EQUIP_TYPE_5_xv501a(
	i1:=NOT sludge_holding_A.q3  OR hold_thickening_process ,
	i2:= sludge_holding_A.q3,
	sa1:=XV505A_SolenoidValveLine_CloseStat ,
	sa2:=XV505A_SolenoidValveLine_OpenStat ,
	c1=> ,
	q1=>XV505A_SolenoidValveLine_OpenCmd ,
	e1=> );
EQUIP_TYPE_5_xv501b(
	i1:=NOT sludge_holding_A.q4  OR hold_thickening_process ,
	i2:= sludge_holding_A.q4,
	sa1:=XV501A_AirBlowerValve_CloseStat ,
	sa2:=XV501A_AirBlowerValve_OpenStat ,
	c1=> ,
	q1=>XV501A_AirBlowerValve_OpenCmd ,
	e1=> );

EQUIP_TYPE_4_d503(
	i1:=NOT sludge_holding_A.q5  OR hold_thickening_process ,
	i2:= sludge_holding_A.q5,
	sa1:= D503A_DrumThickener_EStopStat,
	sa2:= D503A_DrumThickener_LocalRemoteStat,
	sa3:= D503A_DrumThickener_OverloadStat,
	sa4:= D503A_DrumThickener_RunStat,
	c1=> ,
	q1=> D503A_DrumThickener_RunCmd );

EQUP_TYPE_1_p505(
	i1:=NOT sludge_holding_A.q6  OR hold_thickening_process ,
	i2:=sludge_holding_A.q6 ,
	r1:=reset_p505 ,
	sa1:= P505A_BackwashWaterPump_EStopStat,
	sa2:= ,
	sa3:= P505A_BackwashWaterPump_LocalRemoteStat,
	sa4:= P505A_BackwashWaterPump_OverloadStat ,
	sa5:= P505A_BackwashWaterPump_RunStat,
	sb1:= P505B_BackwashWaterPump_EStopStat,
	sb2:= ,
	sb3:= P505B_BackwashWaterPump_LocalRemoteStat,
	sb4:= P505B_BackwashWaterPump_OverloadStat ,
	sb5:= P505B_BackwashWaterPump_RunStat,
	c1=> ,
	c2=> ,
	q1=>P505A_BackwashWaterPump_RunCmd ,
	q2=>P505B_BackwashWaterPump_RunCmd ,
	e1=> );

EQUIP_TYPE_5_xv505A(
	i1:=NOT sludge_holding_A.q7  OR hold_thickening_process ,
	i2:=sludge_holding_A.q7 ,
	sa1:= XV505A_SolenoidValveLine_CloseStat,
	sa2:= XV505A_SolenoidValveLine_OpenStat,
	c1=> ,
	q1=> XV505A_SolenoidValveLine_OpenCmd,
	e1=> );
EQUIP_TYPE_5_xv505B(
	i1:=NOT sludge_holding_A.q7  OR hold_thickening_process ,
	i2:=sludge_holding_A.q7 ,
	sa1:= XV505B_SolenoidValveLine_CloseStat,
	sa2:= XV505B_SolenoidValveLine_OpenStat,
	c1=> ,
	q1=> XV505B_SolenoidValveLine_CloseCmd,
	e1=> );
EQUIP_TYPE_4_M502A(
	i1:= NOT sludge_holding_A.q8  OR hold_thickening_process,
	i2:= sludge_holding_A.q8,
	sa1:= M502A_Floculator_EStopStat,
	sa2:= M502A_Floculator_LocalRemoteStat,
	sa3:= M502A_Floculator_OverloadStat,
	sa4:= M502A_Floculator_RunStat,
	c1=> ,
	q1=> M502A_Floculator_RunCmd,
	e1=> );
EQUIP_TYPE_4_M502B(
	i1:= NOT sludge_holding_A.q8  OR hold_thickening_process,
	i2:= sludge_holding_A.q8,
	sa1:= M502B_Floculator_EStopStat,
	sa2:= M502B_Floculator_LocalRemoteStat,
	sa3:= M502B_Floculator_OverloadStat,
	sa4:= M502B_Floculator_RunStat,
	c1=> ,
	q1=> M502B_Floculator_RunCmd,
	e1=> );

EQUIPMENT_REDUNDANT_AIRBLOWER_p501(
	i1:= sludge_holding_A.q9_1A  OR hold_thickening_process ,
	i2:= sludge_holding_A.q9_2A,
	i3:= sludge_holding_A.q9_1B  OR hold_thickening_process,
	i4:= sludge_holding_A.q9_2B,
	sa1:= P501A_SludgeFeedPump_EStopStat ,
	sa2:= P501A_SludgeFeedPump_IncompleteStat,
	sa3:= P501A_SludgeFeedPump_LocalRemoteStat,
	sa4:= P501A_SludgeFeedPump_OverloadStat,
	sa5:= P501A_SludgeFeedPump_RunStat,
	sb1:= P501B_SludgeFeedPump_EStopStat ,
	sb2:= P501B_SludgeFeedPump_IncompleteStat,
	sb3:= P501B_SludgeFeedPump_LocalRemoteStat,
	sb4:= P501B_SludgeFeedPump_OverloadStat,
	sb5:= P501B_SludgeFeedPump_RunStat,
	sc1:= P501C_SludgeFeedPump_EStopStat ,
	sc2:= P501C_SludgeFeedPump_IncompleteStat,
	sc3:= P501C_SludgeFeedPump_LocalRemoteStat,
	sc4:= P501C_SludgeFeedPumpOverloadStat,
	sc5:= P501C_SludgeFeedPump_RunStat,
	r1 := reset_p501,
	q1=> P501A_SludgeFeedPump_RunCmd,
	q2=> P501B_SludgeFeedPump_RunCmd,
	q3=> P501C_SludgeFeedPump_RunCmd,
	e1=>);

EQUIP_TYPE_5_XVPolymerWaterSupply(
	i1:= sludge_holding_A.q10  OR hold_thickening_process,
	i2:= sludge_holding_A.q11,
	sa1:= XVW501A_WaterValve_CloseStat,
	sa2:= XVW501A_WaterValve_OpenStat ,
	c1=> ,
	q1=> XVW501A_WaterValve_OpenCmd,
	e1=> );

EQUIP_STIRRER_M503(
	i1:= NOT sludge_holding_A.q12  OR hold_thickening_process,
	i2:= sludge_holding_A.q12,
	sa1:= M503_PolymerStirrer_EStopStat,
	sa2:= M503_PolymerStirrer_LocalRemoteStat,
	sa3:= M503_PolymerStirrer_OverloadStat,
	sa4:= M503_PolymerStirrer_RunStat,
	c1=> ,
	q1=>M503_PolymerStirrer_FwdCmd ,
	q2=>M503_PolymerStirrer_RvsCmd ,
	e1=> );

EQUIP_TYPE_1_P602(
	i1:= sludge_holding_A.pfa1 OR hold_inlet_a  OR hold_thickening_process,
	i2:= sludge_holding_A.pfa1,
	r1:= reset_P602,
	sa1:=  P602A_FiltratePump_EStopStat,
	sa2:= ,
	sa3:=  P602A_FiltratePump_LocalRemoteStat,
	sa4:=  P602A_FiltratePump_TripStat ,
	sa5:=  P602A_FiltratePump_RunStat,
	sb1:= P602B_FiltratePump_EStopStat,
	sb2:= ,
	sb3:= P602B_FiltratePump_LocalRemoteStat,
	sb4:= P602A_FiltratePump_TripStat,
	sb5:= P602A_FiltratePump_RunStat ,
	c1=> ,
	c2=> , 
	q1=> P602A_FiltratePump_RunCmd ,
	q2=> P602B_FiltratePump_RunCmd,
	e1=> );

reset_B501 := reset_p505 := reset_p501 := reset_P602 := RST005_ResetButtonSludgeThickening;
END_ACTION
ACTION inlet_mixer:
(*INLET A*)
INLET_A(
	i1:= LSL101A_EQFloatSensor,
	i3:= LSHH103A_SBRFloatSensor,
	i2:= LSH101A_EQFloatSensor,
	i4:= LSHH105A2_StreamLineOverflow,
	i5:= LSL100A_MixerFloatSensor,
	i6:= LSH100A_MixerFloatSensor,
	r1:= rA1,
	i7:= PS101A1_Penstock_OpenStat,
	i8:= PS101A2_Penstock_OpenStat,
	i10:= LSHH105A2_StreamLineOverflow,
	i11:= LSH105A1_StreamLineFlow,
	s1:= F101A1_FineScr_EStopStat,
	s2:= F101A1_FineScr_OverloadStat,
	s3:=F101A2_FineScr_EStopStat ,
	s4:=F101A2_FineScr_OverloadStat ,
	i12:=LSL103A_SBRFloatSensor ,
	i13:=LSH103A_SBRFloatSensor,
	i14:=XV205A_SBRValveR1_OpenStat OR XV206A_SBRValveR2_OpenStat OR XV207A_SBRValveR3_OpenStat OR XV208A_SBRValveR4_OpenStat );

EQUIP_TYPE_1_EQA(
	i1:=INLET_A.q1 ,
	i2:= INLET_A.q2,
	r1:= r_eqA1,
	sa1:= P101A1_EQPump_EStopStat ,
	sa2:= P101A1_EQPump_IncompleteStat ,
	sa3:= P101A1_EQPump_LocalRemoteStat ,
	sa4:= P101A1_EQPump_OverloadStat ,
	sa5:= P101A1_EQPump_RunStat,
	sb1:= P101A2_EQPump_EStopStat ,
	sb2:= P101A2_EQPump_IncompleteStat ,
	sb3:= P101A2_EQPump_LocalRemoteStat,
	sb4:= P101A2_EQPump_OverloadStat  ,
	sb5:= P101A2_EQPump_RunStat,
	c1=> ,
	c2=> ,
	q1=>P101A1_EQPump_RunCmd ,
	q2=>P101A2_EQPump_RunCmd ,
	e1=> );

EQUIP_TYPE_2_MXA(
	i1:= INLET_A.q3,
	i2:= INLET_A.q4,
	sa1:= M101A1_EQMixer_EStopStat,
	sa2:= M101A1_EQMixer_IncompleteStat,
	sa3:= M101A1_EQMixer_LocalRemoteStat,
	sa4:= M101A1_EQMixer_OverloadStat,
	sa5:= M101A1_EQMixer_RunStat,
	sb1:= M101A2_EQMixer_EStopStat,
	sb2:= M101A2_EQMixer_IncompleteStat,
	sb3:= M101A2_EQMixer_LocalRemoteStat,
	sb4:= M101A2_EQMixer_OverloadStat,
	sb5:= M101A2_EQMixer_RunStat,
	c1=> ,
	q1=> M101A1_EQMixer_RunCmd,
	q2=> M101A2_EQMixer_RunCmd,
	e1=> );

EQUIP_TYPE_3_PSA1(
	i1:= NOT INLET_A.q5,
	i2:= INLET_A.q5,
	s1:=PS101A1_Penstock_CloseStat ,
	s2:= PS101A1_Penstock_LocalRemoteStat,
	s3:=PS101A1_Penstock_OpenStat ,
	s4:=PS101A1_Penstock_TripStat ,
	c1=> ,
	q1=>PS101A1_Penstock_CloseCmd ,
	q2=>PS101A1_Penstock_OpenCmd );


EQUIP_TYPE_3_PSA2(
	i1:= NOT INLET_A.q6,
	i2:= INLET_A.q6,
	s1:=PS101A2_Penstock_CloseStat ,
	s2:= PS101A2_Penstock_LocalRemoteStat,
	s3:=PS101A2_Penstock_OpenStat ,
	s4:=PS101A2_Penstock_TripStat ,
	c1=> ,
	q1=>PS101A2_Penstock_CloseCmd ,
	q2=>PS101A2_Penstock_OpenCmd );

EQUIP_TYPE_4_SPA(
	i1:= INLET_A.q9,
	i2:=INLET_A.q10 ,
	sa1:=C101A_ScreenCompactor_EStopStat ,
	sa2:= C101A_ScreenCompactor_LocalRemoteStat,
	sa3:= C101A_ScreeningCompactor_OverloadStat,
	sa4:= C101A_ScreenCompactor_RunStat,
	c1=> ,
	q1=> C101A_ScreenCompactor_RunCmd,
	e1=> );

EQUIP_TYPE_4_SCA(
	i1:=INLET_A.q7,
	i2:= INLET_A.q8,
	sa1:= C102A_ScreenConveyer_EStopStat,
	sa2:= C102A_ScreenConveyer_LocalRemoteStat,
	sa3:= C102A_ScreeningConveyer_OverloadStat,
	sa4:= C102A_ScreenConveyer_RunStat,
	c1=> ,
	q1=> C102A_ScreenConveyer_RunCmd,
	e1=> );

EQUIP_TYPE_5_CWSA(
	i1:=INLET_A.q11 ,
	i2:=INLET_A.q12 ,
	sa1:= XV102A1_ContinuosValveWater_CloseStat,
	sa2:=XV102A1_ContinuosValveWater_OpenStat ,
	c1=> ,
	q1=> XV102A1_ContinuosValveWater_OpenCmd,
	e1=> );

EQUIP_TYPE_4_FSA1(
	i1:= INLET_A.q13,
	i2:= INLET_A.q14,
	sa1:= F101A1_FineScr_EStopStat,
	sa2:= F101A1_FineScr_LocalRemoteStat,
	sa3:= F101A1_FineScr_OverloadStat,
	sa4:= F101A1_FineScr_RunStat,
	c1=> ,
	q1=> F101A1_FineScr_RunCmd,
	e1=> );


EQUIP_TYPE_4_FSA2(
	i1:= INLET_A.q15,
	i2:= INLET_A.q16,
	sa1:= F101A2_FineScr_EStopStat,
	sa2:= F101A2_FineScr_LocalRemoteStat,
	sa3:= F101A2_FineScr_OverloadStat,
	sa4:= F101A2_FineScr_RunStat,
	c1=> ,
	q1=> F101A2_FineScr_RunCmd,
	e1=> );


EQUIP_TYPE_6_WSA1(
	i1:=INLET_A.q17 ,
	i2:=INLET_A.q18 ,
	sa1:=XV101A1_SolenoidValveSpray_CloseStat ,
	sa2:=XV101A1_SolenoidValveSpray_OpenStat ,
	c1=> ,
	q1=>XV101A1_SolenoidValveSpray_OpenCmd ,
	e1=> );

EQUIP_TYPE_6_WSA2(
	i1:=INLET_A.q19 ,
	i2:=INLET_A.q20 ,
	sa1:=XV101A2_SolenoidValveSpray_CloseStat ,
	sa2:=XV101A2_SolenoidValveSpray_OpenStat ,
	c1=> ,
	q1=>XV101A2_SolenoidValveSpray_OpenCmd ,
	e1=> );

EQUIP_TYPE_5_GRVA1(
	i1:=NOT INLET_A.q21 ,
	i2:=INLET_A.q21 ,
	sa1:=XV100A1_GritRemovalValve_CloseStat ,
	sa2:=XV100A1_GritRemovalValve_OpenStat ,
	c1=> XV100A1_GritRemovalValve_OpenCmd,
	q1=> ,
	e1=> );


EQUIP_TYPE_5_GRVA2(
	i1:=NOT INLET_A.q22 ,
	i2:=INLET_A.q22 ,
	sa1:=XV100A2_GritRemovalValve_CloseStat ,
	sa2:=XV100A2_GritRemovalValve_OpenStat ,
	c1=> XV100A1_GritRemovalValve_OpenCmd,
	q1=> ,
	e1=> );


EQUIP_TYPE_4_ClassifierA(
	i1:=INLET_A.q25 ,
	i2:=INLET_A.q26 ,
	sa1:=C103A_GritClasifier_EStopStat ,
	sa2:= C103A_GritClasifier_LocalRemoteStat,
	sa3:= C103A_GritClasifier_RunStat,
	sa4:= C103A_GritClassifier_OverloadStat,
	c1=> ,
	q1=>C103A_GritClasifier_RunCmd ,
	e1=> );

EQUP_TYPE_1_STA1(
	i1:=INLET_A.q27 ,
	i2:=INLET_A.q28 ,
	r1:=r_STA1 ,
	sa1:=P102A1_SBRTransferPump_EStopStat ,
	sa2:=P102A1_SBRTransferPump_IncompleteStat ,
	sa3:=P102A1_SBRTransferPump_LocalRemoteStat ,
	sa4:=P102A1_SBRTransferPump_OverloadStat ,
	sa5:=P102A1_SBRTransferPump_RunStat ,
	sb1:=P102A2_SBRTransferPump_EStopStat ,
	sb2:=P102A2_SBRTransferPump_IncompleteStat ,
	sb3:=P102A2_SBRTransferPump_LocalRemoteStat ,
	sb4:=P102A2_SBRTransferPump_OverloadStat ,
	sb5:=P102A2_SBRTransferPump_RunStat ,
	c1=> ,
	c2=> ,
	q1=>P102A1_SBRTransferPump_RunCmd ,
	q2=>P102A2_SBRTransferPump_RunCmd ,
	e1=> );



IF NOT hold_inlet_b THEN
(* INLET B *)
INLET_B(
	i1:= LSL101B_EQFloatSensor,
	i3:= LSHH103B_SBRFloatSensor,
	i2:= LSH101B_EQFloatSensor,
	i4:= LSHH105B2_StreamLineOverflow,
	i5:= LSL100B_MixerFloatSensor,
	i6:= LSH100B_MixerFloatSensor,
	r1:= rB1,
	i7:= PS101B1_Penstock_OpenStat,
	i8:= PS101B2_Penstock_OpenStat,
	i10:= LSHH105B2_StreamLineOverflow,
	i11:= LSH105B1_StreamLineFlow,
	s1:= F101B1_FineScr_EStopStat,
	s2:= F101B1_FineScr_OverloadStat,
	s3:=F101B2_FineScr_EStopStat ,
	s4:=F101B2_FineScr_OverloadStat ,
	i12:=LSL103B_SBRFloatSensor ,
	i13:=LSH103B_SBRFloatSensor ,
	i14:=XV205B_SBRValveR1_OpenStat OR XV206B_SBRValveR2_OpenStat OR XV207B_SBRValveR3_OpenStat OR XV208B_SBRValveR4_OpenStat );
END_IF

EQUIP_TYPE_1_EQB(
	i1:=INLET_B.q1 OR hold_inlet_b ,
	i2:= INLET_B.q2,
	r1:= r_eqB1,
	sa1:= P101B1_EQPump_EStopStat ,
	sa2:= P101B1_EQPump_IncompleteStat ,
	sa3:= P101B1_EQPump_LocalRemoteStat ,
	sa4:= P101B1_EQPump_OverloadStat ,
	sa5:= P101B1_EQPump_RunStat,
	sb1:= P101B2_EQPump_EStopStat ,
	sb2:= P101B2_EQPump_IncompleteStat ,
	sb3:= P101B2_EQPump_LocalRemoteStat,
	sb4:= P101B2_EQPump_OverloadStat  ,
	sb5:= P101B2_EQPump_RunStat,
	c1=> ,
	c2=> ,
	q1=>P101B1_EQPump_RunCmd ,
	q2=>P101B2_EQPump_RunCmd ,
	e1=> );

EQUIP_TYPE_2_MXB(
	i1:= INLET_B.q3  OR hold_inlet_b,
	i2:= INLET_B.q4,
	sa1:= M101B1_EQMixer_EStopStat,
	sa2:= M101B1_EQMixer_IncompleteStat,
	sa3:= M101B1_EQMixer_LocalRemoteStat,
	sa4:= M101B1_EQMixer_OverloadStat,
	sa5:= M101B1_EQMixer_RunStat,
	sb1:= M101B2_EQMixer_EStopStat,
	sb2:= M101B2_EQMixer_IncompleteStat,
	sb3:= M101B2_EQMixer_LocalRemoteStat,
	sb4:= M101B2_EQMixer_OverloadStat,
	sb5:= M101B2_EQMixer_RunStat,
	c1=> ,
	q1=> M101B1_EQMixer_RunCmd,
	q2=> M101B2_EQMixer_RunCmd,
	e1=> );

EQUIP_TYPE_3_PSB1(
	i1:= NOT INLET_B.q5  OR hold_inlet_b,
	i2:= INLET_B.q5,
	s1:=PS101B1_Penstock_CloseStat ,
	s2:= PS101B1_Penstock_LocalRemoteStat,
	s3:=PS101B1_Penstock_OpenStat ,
	s4:=PS101B1_Penstock_TripStat ,
	c1=> ,
	q1=>PS101B1_Penstock_CloseCmd ,
	q2=>PS101B1_Penstock_OpenCmd );


EQUIP_TYPE_3_PSB2(
	i1:= NOT INLET_B.q6  OR hold_inlet_b,
	i2:= INLET_B.q6,
	s1:=PS101B2_Penstock_CloseStat ,
	s2:= PS101B2_Penstock_LocalRemoteStat,
	s3:=PS101B2_Penstock_OpenStat ,
	s4:=PSB101B2_Penstock_TripStat,
	c1=> ,
	q1=>PS101B2_Penstock_CloseCmd ,
	q2=>PS101B2_Penstock_OpenCmd );

EQUIP_TYPE_4_SPB(
	i1:= INLET_B.q9  OR hold_inlet_b,
	i2:=INLET_B.q10 ,
	sa1:=C101B_ScreenCompactor_EStopStat ,
	sa2:= C101B_ScreenCompactor_LocalRemoteStat,
	sa3:= C101B_ScreeningCompactor_OverloadStat,
	sa4:= C101B_ScreenCompactor_RunStat,
	c1=> ,
	q1=> C101B_ScreenCompactor_RunCmd,
	e1=> );

EQUIP_TYPE_4_SCB(
	i1:=INLET_B.q7  OR hold_inlet_b,
	i2:= INLET_B.q8,
	sa1:= C102B_ScreenConveyer_EStopStat,
	sa2:= C102B_ScreenConveyer_LocalRemoteStat,
	sa3:= C102B_ScreeningConveyer_OverloadStat,
	sa4:= C102B_ScreenConveyer_RunStat,
	c1=> ,
	q1=> C102B_ScreenConveyer_RunCmd,
	e1=> );

EQUIP_TYPE_5_CWSB(
	i1:=INLET_B.q11  OR hold_inlet_b ,
	i2:=INLET_B.q12 ,
	sa1:= XV102B1_ContinuosValveWater_CloseStat,
	sa2:=XV102B1_ContinuosValveWater_OpenStat ,
	c1=> ,
	q1=> XV102B1_ContinuosValveWater_OpenCmd,
	e1=> );

EQUIP_TYPE_4_FSB1(
	i1:= INLET_B.q13  OR hold_inlet_b,
	i2:= INLET_B.q14,
	sa1:= F101B1_FineScr_EStopStat,
	sa2:= F101B1_FineScr_LocalRemoteStat,
	sa3:= F101B1_FineScr_OverloadStat,
	sa4:= F101B1_FineScr_RunStat,
	c1=> ,
	q1=> F101B1_FineScr_RunCmd,
	e1=> );


EQUIP_TYPE_4_FSB2(
	i1:= INLET_B.q15  OR hold_inlet_b,
	i2:= INLET_B.q16,
	sa1:= F101B2_FineScr_EStopStat,
	sa2:= F101B2_FineScr_LocalRemoteStat,
	sa3:= F101B2_FineScr_OverloadStat,
	sa4:= F101B2_FineScr_RunStat,
	c1=> ,
	q1=> F101B2_FineScr_RunCmd,
	e1=> );


EQUIP_TYPE_6_WSB1(
	i1:=INLET_B.q17  OR hold_inlet_b ,
	i2:=INLET_B.q18 ,
	sa1:=XV101B1_SolenoidValveSpray_CloseStat ,
	sa2:=XV101B1_SolenoidValveSpray_OpenStat ,
	c1=> ,
	q1=>XV101B1_SolenoidValveSpray_OpenCmd ,
	e1=> );

EQUIP_TYPE_6_WSB2(
	i1:=INLET_B.q19  OR hold_inlet_b ,
	i2:=INLET_B.q20 ,
	sa1:=XV101B2_SolenoidValveSpray_CloseStat ,
	sa2:=XV101B2_SolenoidValveSpray_OpenStat ,
	c1=> ,
	q1=>XV101B2_SolenoidValveSpray_OpenCmd ,
	e1=> );

EQUIP_TYPE_5_GRVB1(
	i1:=NOT INLET_B.q21  OR hold_inlet_b ,
	i2:=INLET_B.q21 ,
	sa1:=XV100B1_GritRemovalValve_CloseStat ,
	sa2:=XV100B1_GritRemovalValve_OpenStat ,
	c1=> XV100B1_GritRemovalValve_OpenCmd,
	q1=> ,
	e1=> );


EQUIP_TYPE_5_GRVB2(
	i1:=NOT INLET_B.q22   OR hold_inlet_b,
	i2:=INLET_B.q22 ,
	sa1:=XV100B2_GritRemovalValve_CloseStat ,
	sa2:=XV100B2_GritRemovalValve_OpenStat ,
	c1=> XV100B1_GritRemovalValve_OpenCmd,
	q1=> ,
	e1=> );


EQUIP_TYPE_4_ClassifierB(
	i1:=INLET_B.q25   OR hold_inlet_b,
	i2:=INLET_B.q26 ,
	sa1:=C103B_GritClasifier_EStopStat ,
	sa2:= C103B_GritClasifiier_LocalRemoteStat,
	sa3:= C103B_GritClassifier_OverloadStat,
	sa4:= C103B_GritClasifier_RunStat,
	c1=> ,
	q1=>C103B_GritClasifier_RunCmd ,
	e1=> );

EQUP_TYPE_1_STB1(
	i1:=INLET_B.q27   OR hold_inlet_b,
	i2:=INLET_B.q28 ,
	r1:=r_STB1 ,
	sa1:=P102B1_SBRTransferPump_EStopStat ,
	sa2:=P102B1_SBRTransferPump_IncompleteStat ,
	sa3:=P102B1_SBRTransferPump_LocalRemoteStat ,
	sa4:=P102B1_SBRTransferPump_OverloadStat ,
	sa5:=P102B1_SBRTransferPump_RunStat ,
	sb1:=P102B2_SBRTransferPump_EStopStat ,
	sb2:=P102B2_SBRTransferPump_IncompleteStat ,
	sb3:=P102B2_SBRTransferPump_LocalRemoteStat ,
	sb4:=P102B2_SBRTransferPump_OverloadStat ,
	sb5:=P102B2_SBRTransferPump_RunStat ,
	c1=> ,
	c2=> ,
	q1=>P102B1_SBRTransferPump_RunCmd ,
	q2=>P102B2_SBRTransferPump_RunCmd ,
	e1=> );


(*EQ blower*)
EQUP_TYPE_7_Blower(
	i1:=INLET_A.q23 AND (INLET_B.q23 AND NOT GenActive) OR ( hold_inlet_b AND hold_inlet_a),
	i2:= INLET_A.q24 OR (INLET_B.q24 AND NOT GenActive),
	r1:=rblower ,
	sa1:= B101A1_AirBlower_EStopStat,
	sa2:= B101A1_AirBlower_IncompleteStat ,
	sa3:= B101A1_AirBlower_LocalRemoteStat,
	sa4:= B101A1_AirBlower_OverloadStat ,
	sa5:= B101A1_AirBlower_OnOffStat,
	sb1:= B101A2_AirBlower_EStopStat,
	sb2:= B101A2_AirBlower_IncompleteStat ,
	sb3:= B101A2_AirBlower_LocalRemoteStat,
	sb4:= B101A2_AirBlower_OverloadStat ,
	sb5:= B101A2_AirBlower_OnOffStat,
	c1=> ,
	c2=> ,
	q1=> B101A1_AirBlower_RunCmd,
	q2=> B101A2_AirBlower_RunCmd,
	e1=> );


 rA1 := r_eqA1 := r_STA1 := RST001A_ResetButtonInlet_1 ;
 rB1 := r_eqB1 := r_STB1 := RST001B_ResetButtonInlet_2 ;
rblower := RST001A_ResetButtonInlet_1 OR RST001B_ResetButtonInlet_2 ;
END_ACTION
ACTION reactorA:
(*REACTOR A*)
IF NOT hold_SBR_A  THEN
reactorA1(
	op:= OPR1A_ReactorStatus,
	res_fill:=Fill_selectorA.q1 AND NOT holdFill_A ,
	i1:= LSH201A1_LevelSensorR1 ,
	alum_time:= Alum_reactorA1,
	res_aeration:= Aerate_selectorA.q1,
	ph1:=PHT201A1_pHlevelR1 ,
	res_decanting:=Decant_selectorA.q1 ,
	r1:=resumeAlumA1 ,
	i2:=LSHH501A_SludgeStorage ,
	i3:=HR201A1_DecantHighLevelR1 ,
	i4:=LR201A1_DecantLowLevelR1 ,
	reset := sbr_reset_A1,
	req_fill=> ,
	q1=> ,
	q2=> ,
	q4=> ,
	q3=> ,
	q5=> ,
	q6=> ,
	req_aeration=> ,
	e1=>alarm_alum_sbr_A1 ,
	q7=> ,
	q8=> ,
	m1=> ,
	req_settle=> ,
	req_decanting=> ,
	q9=> );

reactorA2(
	op:= OPR2A_ReactorStatus,
	res_fill:=Fill_selectorA.q2 AND NOT holdFill_A  ,
	i1:= LSH201A2_LevelSensorR2 ,
	alum_time:= Alum_reactorA2,
	res_aeration:= Aerate_selectorA.q2,
	ph1:=PHT201A2_pHlevelR2 ,
	res_decanting:=Decant_selectorA.q2 ,
	r1:=resumeAlumA2 ,
	i2:=LSHH501A_SludgeStorage ,
	i3:=HR201A2_DecantHighLevelR2 ,
	i4:=LR201A2_DecantLowLevelR2 ,
	reset := sbr_reset_A2,
	req_fill=> ,
	q1=> ,
	q2=> ,
	q4=> ,
	q3=> ,
	q5=> ,
	q6=> ,
	req_aeration=> ,
	e1=>alarm_alum_sbr_A2 ,
	q7=> ,
	q8=> ,
	m1=> ,
	req_settle=> ,
	req_decanting=> ,
	q9=> );

reactorA3(
	op:= OPR3A_ReactorStatus,
	res_fill:=Fill_selectorA.q3 AND NOT holdFill_A  ,
	i1:= LSH201A3_LevelSensorR3 ,
	alum_time:= Alum_reactorA3,
	res_aeration:= Aerate_selectorA.q3,
	ph1:=PHT201A3_pHlevelR3 ,
	res_decanting:=Decant_selectorA.q3 ,
	r1:=resumeAlumA3 ,
	i2:=LSHH501A_SludgeStorage ,
	i3:=HR201A3_DecantHighLevelR3 ,
	i4:=LR201A3_DecantLowLevelR3 ,
	reset := sbr_reset_A3,
	req_fill=> ,
	q1=> ,
	q2=> ,
	q4=> ,
	q3=> ,
	q5=> ,
	q6=> ,
	req_aeration=> ,
	e1=>alarm_alum_sbr_A3 ,
	q7=> ,
	q8=> ,
	m1=> ,
	req_settle=> ,
	req_decanting=> ,
	q9=> );

reactorA4(
	op:= OPR4A_ReactorStatus,
	res_fill:=Fill_selectorA.q4  AND NOT holdFill_A ,
	i1:= LSH201A4_LevelSensorR4 ,
	alum_time:= Alum_reactorA4,
	res_aeration:= Aerate_selectorA.q4,
	ph1:=PHT201A4_pHlevelR4 ,
	res_decanting:=Decant_selectorA.q4 ,
	r1:=resumeAlumA4 ,
	i2:=LSHH501A_SludgeStorage ,
	i3:=HR201A4_DecantHighLevelR4 ,
	i4:=LR201A4_DecantLowLevelR4 ,
	reset := sbr_reset_A4,
	req_fill=> ,
	q1=> ,
	q2=> ,
	q4=> ,
	q3=> ,
	q5=> ,
	q6=> ,
	req_aeration=> ,
	e1=>alarm_alum_sbr_A4 ,
	q7=> ,
	q8=> ,
	m1=> ,
	req_settle=> ,
	req_decanting=> ,
	q9=> );

fill_selectorA(
	i1:=ReactorA1.req_fill ,
	i2:=ReactorA2.req_fill ,
	i3:=ReactorA3.req_fill ,
	i4:=ReactorA4.req_fill,
	q1=> ,
	q2=> ,
	q3=> ,
	q4=> ,
	c1=> );

aerate_selectorA(
	i1:=ReactorA1.req_aeration,
	i2:=ReactorA2.req_aeration ,
	i3:=ReactorA3.req_aeration ,
	i4:=ReactorA4.req_aeration ,
	available:=2 ,
	q1=> ,
	q2=> ,
	q3=> ,
	q4=>);

decant_selectorA(
	i1:=  ReactorA1.req_decanting,
	i2:=  ReactorA2.req_decanting,
	i3:=  ReactorA3.req_decanting,
	i4:=  ReactorA4.req_decanting,
	q1=> ,
	q2=> ,
	q3=> ,
	q4=> ,
	c1=> );
END_IF

sbr_airblower_A(
	hold := hold_SBR_A,
	sa1:= B201A1_AirBlowerS1_EStopStat,
	sa2:= B201A1_AirBlowerS1_IncompleteStat,
	sa3:= B201A1_AirBlowerS1_LocalRemoteStat,
	sa4:= B201A1_AirBlowerS1_OverloadStat,
	sa5:= B201A1_AirBlowerS1_RunStat,
	sb1:= B201A2_AirBlowerS1_EStopStat,
	sb2:= B201A2_AirBlowerS1_IncompleteStat,
	sb3:= B201A2_AirBlowerS1_LocalRemoteStat,
	sb4:= B201A2_AirBlowerS1_OverloadStat,
	sb5:= B201A2_AirBlowerS1_RunStat,
	sc1:= B201A3_AirBlowerS1_EStopStat,
	sc2:= B201A3_AirBlowerS1_IncompleteStat,
	sc3:= B201A3_AirBlowerS1_LocalRemoteStat,
	sc4:= B201A3_AirBlowerS1_OverloadStat,
	sc5:= B201A3_AirBlowerS1_RunStat,
	req:= aerate_selectorA.taken,
	rq1=> B201A1_AirBlowerS1_RunCmd,
	rq2=> B201A2_AirBlowerS1_RunCmd,
	rq3=> B201A3_AirBlowerS1_RunCmd);


EQUP_TYPE_1_Pump_RA(
	i1:= NOT( reactorA1.q6 AND reactorA2.q6 AND reactorA3.q6 AND reactorA4.q6) OR hold_desludging_A OR hold_SBR_A,
	i2:= (reactorA1.q6 OR reactorA2.q6 OR reactorA3.q6 OR reactorA4.q6) ,
	r1:= reset_Pump2_RA,
	sa1:=P201A1_DesludgePumpS1_EStopStat ,
	sa2:= ,
	sa3:=P201A1_DesludgePumpS1_LocalRemoteStat ,
	sa4:= P201A1_DesludgePumpS1_OverloadStatus,
	sa5:=P201A1_DesludgePumpS1_RunStat ,
	sb1:= P201A2_DesludgePumpS1_EStopStat,
	sb2:= ,
	sb3:=P201A2_DesludgePumpS1_LocalRemoteStat ,
	sb4:= P201A2_DesludgePumpS1_OverloadStatus,
	sb5:=P201A2_DesludgePumpS1_RunStat ,
	c1=> ,
	c2=> ,
	q1=>P201A1_DesludgePump_RunCmd,
	q2=>P201A2_DesludgePump_RunCmd ,
	e1=> );


EQUIP_TYPE_3_Valva1_RA1(
	i1:=NOT reactorA1.q1 OR hold_SBR_A,
	i2:=reactorA1.q1 ,
	s1:=XV205A_SBRValveR1_CloseStat ,
	s2:=XV205A_SBRValveR1_OpenStat ,
	c1=> ,
	q1=>XV205A_SBRValveR1_CloseCmd ,
	q2=>XV205A_SBRValveR1_OpenCmd);

EQUIP_TYPE_8_MIXER_A1(
	i1:= NOT reactorA1.q2 OR hold_SBR_A,
	i2:= reactorA1.q2,
	sa1:=M200A1A_MixerR1_EStopStat,
	sa2:=M200A1A_MixerR1_IncompleteStat ,
	sa3:=M200A1A_MixerR1_LocalRemoteStat ,
	sa4:=M200A1A_MixerR1_OverloadStat ,
	sa5:=M200A1A_MixerR1_RunStat ,
	sb1:=M200A1B_MixerR1_EStopStat,
	sb2:=M200A1B_MixerR1_IncompleteStat ,
	sb3:=M200A1B_MixerR1_LocalRemoteStat ,
	sb4:=M200A1B_MixerR1_OverloadStat ,
	sb5:=M200A1B_MixerR1_RunStat ,
	sc1:=M200A1C_MixerR1_EStopStat,
	sc2:=M200A1C_MixerR1_IncompleteStat ,
	sc3:=M200A1C_MixerR1_LocalRemoteStat ,
	sc4:=M200A1C_MixerR1_OverloadStat ,
	sc5:=M200A1C_MixerR1_RunStat ,
	c1=> ,
	q1=>M200A1A_MixerR1_RunCmd ,
	q2=>M200A1B_MixerR1_RunCmd,
	q3=>M200A1C_MixerR1_RunCmd ,
	e1=> );

EQUIP_TYPE_3_Valve2_RA1(
	i1:=NOT reactorA1.q3 OR hold_SBR_A,
	i2:= reactorA1.q3,
	s1:= XV221A_LimeValveR1_CloseStat,
	s2:= XV221A_LimeValveR1_OpenStat,
	c1=> ,
	q1=>XV221A_LimeValveR1_CloseCmd ,
	q2=>XV221A_LimeValveR1_OpenCmd );

EQUIP_TYPE_3_Valve3_RA1(
	i1:=NOT reactorA1.q4 OR hold_SBR_A ,
	i2:= reactorA1.q4,
	s1:= XV211A_AlumValveR1_CloseStat,
	s2:= XV211A_AlumValveR1_OpenStat,
	c1=> ,
	q1=>XV211A_AlumValveR1_CloseCmd ,
	q2=>XV211A_AlumValveR1_OpenCmd );

EQUIP_TYPE_3_Valve4_RA1(
	i1:=NOT reactorA1.q5 OR hold_SBR_A ,
	i2:= reactorA1.q5,
	s1:=XV201A_AirBlowerValveR1_CloseStat ,
	s2:=XV201A_AirBlowerValveR1_OpenStat ,
	c1=> ,
	q1=>XV201A_AirBlowerValveR1_CloseCmd ,
	q2=>XV201A_AirBlowerValveR1_OpenCmd );

EQUIP_TYPE_9_Valve5_RA1(
	i1:= NOT reactorA1.q7  OR hold_SBR_A,
	i2:=reactorA1.q7 ,
	s1:=XV241A_SludgeValveR1_CloseStat ,
	s2:=XV241A_SludgeValveR1_OpenStat ,
	c1=> ,
	q1=>XV241A_SludgeValveR1_CloseCmd ,
	q2=>XV241A_SludgeValveR1_OpenCmd );

EQUIP_TYPE_10_Dec_RA1(
	i1:=reactorA1.q8 OR hold_SBR_A ,
	i2:= reactorA1.q9 OR hold_SBR_A,
	r1:= reset_dec_RA1,
	s1:= XV261A_DecanterR1_EStopStat,
	s2:= XV261A_DecanterR1_FwdStat,
	s3:= XV261A_DecanterR1_OverloadStat,
	s4:= XV261A_DecanterR1_OverloadStat,
	s5:= XV261A_DecanterR1_RvsStat,
	q1=> XV261A_DecanterR1_RvsCmd,
	q2=>XV261A_DecanterR1_FwdCmd ,
	e1=> );




EQUIP_TYPE_3_Valva1_RA2(
	i1:=NOT reactorA2.q1 OR hold_SBR_A ,
	i2:=reactorA2.q1 ,
	s1:=XV206A_SBRValveR2_CloseStat ,
	s2:=XV206A_SBRValveR2_OpenStat ,
	c1=> ,
	q1=>XV206A_SBRValveR2_CloseCmd ,
	q2=>XV206A_SBRValveR2_OpenCmd);

EQUIP_TYPE_8_MIXER_A2(
	i1:= NOT reactorA2.q2 OR hold_SBR_A,
	i2:= reactorA2.q2,
	sa1:=M200A2A_MixerR2_EStopStat,
	sa2:=M200A2A_MixerR2_IncompleteStat ,
	sa3:=M200A2A_MixerR2_LocalRemoteStat ,
	sa4:=M200A2A_MixerR2_OverloadStat ,
	sa5:=M200A2A_MixerR2_RunStat ,
	sb1:=M200A2B_MixerR2_EStopStat,
	sb2:=M200A2B_MixerR2_IncompleteStat ,
	sb3:=M200A2B_MixerR2_LocalRemoteStat ,
	sb4:=M200A2B_MixerR2_OverloadStat ,
	sb5:=M200A2B_MixerR2_RunStat ,
	sc1:=M200A2C_MixerR2_EStopStat,
	sc2:=M200A2C_MixerR2_IncompleteStat ,
	sc3:=M200A2C_MixerR2_LocalRemoteStat ,
	sc4:=M200A2C_MixerR2_OverloadStat ,
	sc5:=M200A2C_MixerR2_RunStat ,
	c1=> ,
	q1=>M200A2A_MixerR2_RunCmd ,
	q2=>M200A2B_MixerR2_RunCmd,
	q3=>M200A2C_MixerR2_RunCmd ,
	e1=> );

EQUIP_TYPE_3_Valve2_RA2(
	i1:=NOT reactorA2.q3 OR hold_SBR_A ,
	i2:= reactorA2.q3,
	s1:= XV222A_LimeValveR2_CloseStat,
	s2:= XV222A_LimeValveR2_OpenStat,
	c1=> ,
	q1=>XV222A_LimeValveR2_CloseCmd ,
	q2=>XV222A_LimeValveR2_OpenCmd );

EQUIP_TYPE_3_Valve3_RA2(
	i1:=NOT reactorA2.q4 OR hold_SBR_A,
	i2:= reactorA2.q4,
	s1:= XV212A_AlumValveR2_CloseStat,
	s2:= XV212A_AlumValveR2_OpenStat,
	c1=> ,
	q1=>XV212A_AlumValveR2_CloseCmd ,
	q2=>XV212A_AlumValveR2_OpenCmd );

EQUIP_TYPE_3_Valve4_RA2(
	i1:=NOT reactorA2.q5 OR hold_SBR_A ,
	i2:= reactorA2.q5,
	s1:=XV202A_AirBlowerValveR2_CloseStat ,
	s2:=XV202A_AirBlowerValveR2_OpenStat ,
	c1=> ,
	q1=>XV202A_AirBlowerValveR2_CloseCmd ,
	q2=>XV202A_AirBlowerValveR2_OpenCmd );


EQUIP_TYPE_9_Valve5_RA2(
	i1:= NOT reactorA2.q7 OR hold_SBR_A ,
	i2:=reactorA2.q7 ,
	s1:=XV242A_SludgeValveR2_CloseStat ,
	s2:=XV242A_SludgeValveR2_OpenStat ,
	c1=> ,
	q1=>XV242A_SludgeValveR2_CloseCmd ,
	q2=>XV242A_SludgeValveR2_OpenCmd );

EQUIP_TYPE_10_Dec_RA2(
	i1:=reactorA2.q8  OR NOT hold_SBR_A,
	i2:= reactorA2.q9 OR NOT hold_SBR_A,
	r1:= reset_dec_RA2,
	s1:= XV262A_DecanterR2_EStopStat,
	s2:= XV262A_DecanterR2_FwdStat,
	s3:= XV262A_DecanterR2_OverloadStat,
	s4:= XV262A_DecanterR2_OverloadStat,
	s5:= XV262A_DecanterR2_RvsStat,
	q1=> XV262A_DecanterR2_RvsCmd,
	q2=>XV262A_DecanterR2_FwdCmd ,
	e1=> );




EQUIP_TYPE_3_Valva1_RA3(
	i1:=NOT reactorA3.q1 OR hold_SBR_A ,
	i2:=reactorA3.q1 ,
	s1:=XV207A_SBRValveR3_CloseStat ,
	s2:=XV207A_SBRValveR3_OpenStat ,
	c1=> ,
	q1=>XV207A_SBRValveR3_CloseCmd ,
	q2=>XV207A_SBRValveR3_OpenCmd);

EQUIP_TYPE_8_MIXER_A3(
	i1:= NOT reactorA3.q2 OR hold_SBR_A,
	i2:= reactorA3.q2,
	sa1:=M200A3A_MixerR3_EStopStat,
	sa2:=M200A3A_MixerR3_IncompleteStat ,
	sa3:=M200A3A_MixerR3_LocalRemoteStat ,
	sa4:=M200A3A_MixerR3_OverloadStat ,
	sa5:=M200A3A_MixerR3_RunStat ,
	sb1:=M200A3B_MixerR3_EStopStat,
	sb2:=M200A3B_MixerR3_IncompleteStat ,
	sb3:=M200A3B_MixerR3_LocalRemoteStat ,
	sb4:=M200A3B_MixerR3_OverloadStat ,
	sb5:=M200A3B_MixerR3_RunStat ,
	sc1:=M200A3C_MixerR3_EStopStat,
	sc2:=M200A3C_MixerR3_IncompleteStat ,
	sc3:=M200A3C_MixerR3_LocalRemoteStat ,
	sc4:=M200A3C_MixerR3_OverloadStat ,
	sc5:=M200A3C_MixerR3_RunStat ,
	c1=> ,
	q1=>M200A3A_MixerR3_RunCmd ,
	q2=>M200A3B_MixerR3_RunCmd,
	q3=>M200A3C_MixerR3_RunCmd ,
	e1=> );

EQUIP_TYPE_3_Valve2_RA3(
	i1:=NOT reactorA3.q3 OR hold_SBR_A,
	i2:= reactorA3.q3,
	s1:= XV223A_LimeValveR3_CloseStat,
	s2:= XV223A_LimeValveR3_OpenStat,
	c1=> ,
	q1=>XV223A_LimeValveR3_CloseCmd ,
	q2=>XV223A_LimeValveR3_OpenCmd );

EQUIP_TYPE_3_Valve3_RA3(
	i1:=NOT reactorA3.q4  OR hold_SBR_A,
	i2:= reactorA3.q4,
	s1:= XV213A_AlumValveR3_CloseStat,
	s2:= XV213A_AlumValveR3_OpenStat,
	c1=> ,
	q1=>XV213A_AlumValveR3_CloseCmd ,
	q2=>XV213A_AlumValveR3_OpenCmd );

EQUIP_TYPE_3_Valve4_RA3(
	i1:=NOT reactorA3.q5 OR hold_SBR_A ,
	i2:= reactorA3.q5,
	s1:=XV203A_AirBlowerValveR3_CloseStat ,
	s2:=XV203A_AirBlowerValveR3_OpenStat ,
	c1=> ,
	q1=>XV203A_AirBlowerValveR3_CloseCmd ,
	q2=>XV203A_AirBlowerValveR3_OpenCmd );


EQUIP_TYPE_9_Valve5_RA3(
	i1:= NOT reactorA3.q7  OR hold_SBR_A,
	i2:=reactorA3.q7 ,
	s1:=XV243A_SludgeValveR3_CloseStat ,
	s2:=XV243A_SludgeValveR3_OpenStat ,
	c1=> ,
	q1=>XV243A_SludgeValveR3_CloseCmd ,
	q2=>XV243A_SludgeValveR3_OpenCmd );

EQUIP_TYPE_10_Dec_RA3(
	i1:=reactorA3.q8 OR NOT  hold_SBR_A ,
	i2:= reactorA3.q9 OR NOT  hold_SBR_A,
	r1:= reset_dec_RA3,
	s1:= XV263A_DecanterR3_EStopStat,
	s2:= XV263A_DecanterR3_FwdStat,
	s3:= XV263A_DecanterR3_OverloadStat,
	s4:= XV263A_DecanterR3_OverloadStat,
	s5:= XV263A_DecanterR3_RvsStat,
	q1=> XV263A_DecanterR3_RvsCmd,
	q2=>XV263A_DecanterR3_FwdCmd ,
	e1=> );



EQUIP_TYPE_3_Valva1_RA4(
	i1:=NOT reactorA4.q1 OR hold_SBR_A ,
	i2:=reactorA4.q1 ,
	s1:=XV208A_SBRValveR4_CloseStat ,
	s2:=XV208A_SBRValveR4_OpenStat ,
	c1=> ,
	q1=>XV208A_SBRValveR4_CloseCmd ,
	q2=>XV208A_SBRValveR4_OpenCmd);

EQUIP_TYPE_8_MIXER_A4(
	i1:= NOT reactorA4.q2 OR hold_SBR_A,
	i2:= reactorA4.q2,
	(*sa1:=M200A4A_MixerR4_EStopStat,*)
	sa2:=M200A4A_MixerR4_IncompleteStat ,
	sa3:=M200A4A_MixerR4_LocalRemoteStat ,
	sa4:=M200A4A_MixerR4_OverloadStat ,
	sa5:=M200A4A_MixerR4_RunStat ,
	(*sb1:=M200A4B_MixerR4_EStopStat,*)
	sb2:=M200A4B_MixerR4_IncompleteStat ,
	sb3:=M200A4B_MixerR4_LocalRemoteStat ,
	sb4:=M200A4B_MixerR4_OverloadStat ,
	sb5:=M200A4B_MixerR4_RunStat ,
	(*sc1:=M200A4C_MixerR4_EStopStat,*)
	sc2:=M200A4C_MixerR4_IncompleteStat ,
	sc3:=M200A4C_MixerR4_LocalRemoteStat ,
	sc4:=M200A4C_MixerR4_OverloadStat ,
	sc5:=M200A4C_MixerR4_RunStat ,
	c1=> ,
	q1=>M200A4A_MixerR4_RunCmd ,
	q2=>M200A4B_MixerR4_RunCmd,
	q3=>M200A4C_MixerR4_RunCmd ,
	e1=> );

EQUIP_TYPE_3_Valve2_RA4(
	i1:=NOT reactorA4.q3 OR hold_tertiary_process OR hold_SBR_A ,
	i2:= reactorA4.q3,
	s1:= XV224A_LimeValveR4_CloseStat,
	s2:= XV224A_LimeValveR4_OpenStat,
	c1=> ,
	q1=>XV224A_LimeValveR4_CloseCmd ,
	q2=>XV224A_LimeValveR4_OpenCmd );

EQUIP_TYPE_3_Valve3_RA4(
	i1:=NOT reactorA4.q4 OR hold_tertiary_process OR hold_SBR_A ,
	i2:= reactorA4.q4,
	s1:= XV214A_AlumValveR4_CloseStat,
	s2:= XV214A_AlumValveR4_OpenStat,
	c1=> ,
	q1=>XV214A_AlumValveR4_CloseCmd ,
	q2=>XV214A_AlumValveR4_OpenCmd );

EQUIP_TYPE_3_Valve4_RA4(
	i1:=NOT reactorA4.q5 OR hold_SBR_A ,
	i2:= reactorA4.q5,
	s1:=XV204A_AirBlowerValveR4_CloseStat ,
	s2:=XV204A_AirBlowerValveR4_OpenStat ,
	c1=> ,
	q1=>XV204A_AirBlowerValveR4_CloseCmd ,
	q2=>XV204A_AirBlowerValveR4_OpenCmd );

EQUIP_TYPE_9_Valve5_RA4(
	i1:= NOT reactorA4.q7 OR hold_SBR_A ,
	i2:=reactorA4.q7 ,
	s1:=XV244A_SludgeValveR4_CloseStat ,
	s2:=XV244A_SludgeValveR4_OpenStat ,
	c1=> ,
	q1=>XV244A_SludgeValveR4_CloseCmd ,
	q2=>XV244A_SludgeValveR4_OpenCmd );

EQUIP_TYPE_10_Dec_RA4(
	i1:=reactorA4.q8 OR  NOT hold_SBR_A ,
	i2:= reactorA4.q9 OR NOT  hold_SBR_A,
	r1:= reset_dec_RA4,
	s1:= XV264A_DecanterR4_EStopStat,
	s2:= XV264A_DecanterR4_FwdStat,
	s3:= XV264A_DecanterR4_OverloadStat,
	s4:= XV264A_DecanterR4_OverloadStat,
	s5:= XV264A_DecanterR4_RvsStat,
	q1=> XV264A_DecanterR4_RvsCmd,
	q2=>XV264A_DecanterR4_FwdCmd ,
	e1=> );

reset_Pump2_RA := reset_dec_RA1 := reset_dec_RA2 := reset_dec_RA3 := reset_dec_RA4 := RST003A_ResetButtonSBR_1;


timeConversion_alumA1(inputTime:=InputTime_alumA1 , atTime:= alum_reactorA1, outputTime=>OutputTime_alumA1 );
timeConversion_alumA2(inputTime:=InputTime_alumA2 , atTime:= alum_reactorA2, outputTime=>OutputTime_alumA2 );
timeConversion_alumA3(inputTime:=InputTime_alumA3 , atTime:= alum_reactorA3, outputTime=>OutputTime_alumA3 );
timeConversion_alumA4(inputTime:=InputTime_alumA4 , atTime:= alum_reactorA4, outputTime=>OutputTime_alumA4 );
END_ACTION
ACTION reactorB:
(*REACTOR A*)
IF NOT hold_SBR_B THEN
reactorB1(
	op:= OPR1B_ReactorStatus,
	res_fill:=Fill_selectorB.q1 AND NOT holdFill_B ,
	i1:= LSH201B1_LevelSensorR1 ,
	alum_time:= Alum_reactorB1,
	res_aeration:= Aerate_selectorB.q1,
	ph1:=PHT201B1_pHlevelR1 ,
	res_decanting:=Decant_selectorB.q1 ,
	r1:=resumeAlumB1 ,
	i2:=LSHH501B_SludgeStorage ,
	i3:=HR201B1_DecantHighLevelR1 ,
	i4:=LR201B1_DecantLowLevelR1 ,
	reset := sbr_reset_B1,
	req_fill=> ,
	q1=> ,
	q2=> ,
	q4=> ,
	q3=> ,
	q5=> ,
	q6=> ,
	req_aeration=> ,
	e1=>alarm_alum_sbr_B1 ,
	q7=> ,
	q8=> ,
	m1=> ,
	req_settle=> ,
	req_decanting=> ,
	q9=> );

reactorB2(
	op:= OPR2B_ReactorStatus,
	res_fill:=Fill_selectorB.q2 AND NOT holdFill_B ,
	i1:= LSH201B2_LevelSensorR2 ,
	alum_time:= Alum_reactorB2,
	res_aeration:= Aerate_selectorB.q2,
	ph1:=PHT201B2_pHlevelR2 ,
	res_decanting:=Decant_selectorB.q2 ,
	r1:=resumeAlumB2 ,
	i2:=LSHH501B_SludgeStorage ,
	i3:=HR201B2_DecantHighLevelR2 ,
	i4:=LR201B2_DecantLowLevelR2 ,
	reset := sbr_reset_B2,
	req_fill=> ,
	q1=> ,
	q2=> ,
	q4=> ,
	q3=> ,
	q5=> ,
	q6=> ,
	req_aeration=> ,
	e1=>alarm_alum_sbr_B2 ,
	q7=> ,
	q8=> ,
	m1=> ,
	req_settle=> ,
	req_decanting=> ,
	q9=> );

reactorB3(
	op:= OPR3B_ReactorStatus,
	res_fill:=Fill_selectorB.q3 AND NOT holdFill_B ,
	i1:= LSH201B3_LevelSensorR3 ,
	alum_time:= Alum_reactorB3,
	res_aeration:= Aerate_selectorB.q3,
	ph1:=PHT201B3_pHlevelR3 ,
	res_decanting:=Decant_selectorB.q3 ,
	r1:=resumeAlumB3 ,
	i2:=LSHH501B_SludgeStorage ,
	i3:=HR201B3_DecantHighLevelR3 ,
	i4:=LR201B3_DecantLowLevelR3 ,
	reset := sbr_reset_B3,
	req_fill=> ,
	q1=> ,
	q2=> ,
	q4=> ,
	q3=> ,
	q5=> ,
	q6=> ,
	req_aeration=> ,
	e1=>alarm_alum_sbr_B3 ,
	q7=> ,
	q8=> ,
	m1=> ,
	req_settle=> ,
	req_decanting=> ,
	q9=> );

reactorB4(
	op:= OPR4B_ReactorStatus,
	res_fill:=Fill_selectorB.q4 AND NOT holdFill_B,
	i1:= LSH201B4_LevelSensorR4 ,
	alum_time:= Alum_reactorB4,
	res_aeration:= Aerate_selectorB.q4,
	ph1:=PHT201B4_pHlevelR4 ,
	res_decanting:=Decant_selectorB.q4 ,
	r1:=resumeAlumB4 ,
	i2:=LSHH501B_SludgeStorage ,
	i3:=HR201B4_DecantHighLevelR4 ,
	i4:=LR201B4_DecantLowLevelR4 ,
	reset := sbr_reset_B4,
	req_fill=> ,
	q1=> ,
	q2=> ,
	q4=> ,
	q3=> ,
	q5=> ,
	q6=> ,
	req_aeration=> ,
	e1=> alarm_alum_sbr_B4,
	q7=> ,
	q8=> ,
	m1=> ,
	req_settle=> ,
	req_decanting=> ,
	q9=> );

fill_selectorB(
	i1:=ReactorB1.req_fill ,
	i2:=ReactorB2.req_fill ,
	i3:=ReactorB3.req_fill ,
	i4:=ReactorB4.req_fill,
	q1=> ,
	q2=> ,
	q3=> ,
	q4=> ,
	c1=> );

aerate_selectorB(
	i1:=ReactorB1.req_aeration,
	i2:=ReactorB2.req_aeration ,
	i3:=ReactorB3.req_aeration ,
	i4:=ReactorB4.req_aeration ,
	available:=2 ,
	q1=> ,
	q2=> ,
	q3=> ,
	q4=>);

decant_selectorB(
	i1:=  ReactorB1.req_decanting,
	i2:=  ReactorB2.req_decanting,
	i3:=  ReactorB3.req_decanting,
	i4:=  ReactorB4.req_decanting,
	q1=> ,
	q2=> ,
	q3=> ,
	q4=> ,
	c1=> );

END_IF


sbr_airblower_B(
	hold := hold_SBR_B,
	sa1:= B201B1_AirBlowerS2_EStopStat,
	sa2:= B201B1_AirBlowerS2_IncompleteStat,
	sa3:= B201B1_AirBlowerS2_LocalRemoteStat,
	sa4:= B201B1_AirBlowerS2_OverloadStat,
	sa5:= B201B1_AirBlowerS2_RunStat,
	sb1:= B201B2_AirBlowerS2_EStopStat,
	sb2:= B201B2_AirBlowerS2_IncompleteStat,
	sb3:= B201B2_AirBlowerS2_LocalRemoteStat,
	sb4:= B201B2_AirBlowerS2_OverloadStat,
	sb5:= B201B2_AirBlowerS2_RunStat,
	sc1:= B201B3_AirBlowerS2_EStopStat,
	sc2:= B201B3_AirBlowerS2_IncompleteStat,
	sc3:= B201B3_AirBlowerS2_LocalRemoteStat,
	sc4:= B201B3_AirBlowerS2_OverloadStat,
	sc5:= B201B3_AirBlowerS2_RunStat,
	req:= aerate_selectorA.taken,
	rq1=> B201B1_AirBlowerS2_RunCmd,
	rq2=> B201B2_AirBlowerS2_RunCmd,
	rq3=> B201B3_AirBlowerS2_RunCmd);


EQUP_TYPE_1_Pump_RB(
	i1:= NOT( reactorB1.q6 AND reactorB2.q6 AND reactorB3.q6 AND reactorB4.q6) OR hold_desludging_B OR hold_SBR_B,
	i2:= (reactorB1.q6 OR reactorB2.q6 OR reactorB3.q6 OR reactorB4.q6),
	r1:= reset_Pump2_RB,
	sa1:=P201B1_DesludgePumpS2_EStopStat ,
	sa2:= ,
	sa3:=P201B1_DesludgePumpS2_LocalRemoteStat ,
	sa4:= P201B1_DesludgePumpS2_OverloadStat,
	sa5:=P201B1_DesludgePumpS2_RunStat ,
	sb1:= P201B2_DesludgePumpS2_EStopStat,
	sb2:= ,
	sb3:=P201B2_DesludgePumpS2_LocalRemoteStat ,
	sb4:= P201B2_DesludgePumpS2_OverloadStat,
	sb5:=P201B2_DesludgePumpS2_RunStat ,
	c1=> ,
	c2=> ,
	q1=>P201B1_DesludgePumpS2_RunCmd,
	q2=>P201B2_DesludgePumpS2_RunCmd ,
	e1=> );


EQUIP_TYPE_3_Valva1_RB1(
	i1:=NOT reactorB1.q1 OR hold_SBR_B ,
	i2:=reactorB1.q1 ,
	s1:=XV205B_SBRValveR1_CloseStat ,
	s2:=XV205B_SBRValveR1_OpenStat ,
	c1=> ,
	q1=>XV205B_SBRValveR1_CloseCmd ,
	q2=>XV205B_SBRValveR1_OpenCmd);

EQUIP_TYPE_8_MIXER_B1(
	i1:= NOT reactorB1.q2 OR hold_SBR_B,
	i2:= reactorB1.q2,
	sa1:=M200B1A_MixerR1_EStopStat,
	sa2:=M200B1A_MixerR1_IncompleteStat ,
	sa3:=M200B1A_MixerR1_LocalRemoteStat ,
	sa4:=M200B1A_MixerR1_OverloadStat ,
	sa5:=M200B1A_MixerR1_RunStat ,
	sb1:=M200B1B_MixerR1_EStopStat,
	sb2:=M200B1B_MixerR1_IncompleteStat ,
	sb3:=M200B1B_MixerR1_LocalRemoteStat ,
	sb4:=M200B1B_MixerR1_OverloadStat ,
	sb5:=M200B1B_MixerR1_RunStat ,
	sc1:=M200B1C_MixerR1_EStopStat,
	sc2:=M200B1C_MixerR1_IncompleteStat ,
	sc3:=M200B1C_MixerR1_LocalRemoteStat ,
	sc4:=M200B1C_MixerR1_OverloadStat ,
	sc5:=M200B1C_MixerR1_RunStat ,
	c1=> ,
	q1=>M200B1A_MixerR1_RunCmd ,
	q2=>M200B1B_MixerR1_RunCmd,
	q3=>M200B1C_MixerR1_RunCmd ,
	e1=> );

EQUIP_TYPE_3_Valve2_RB1(
	i1:=NOT reactorB1.q3 OR hold_tertiary_process OR hold_SBR_B ,
	i2:= reactorB1.q3,
	s1:= XV221B_LimeValveR1_CloseStat,
	s2:= XV221B_LimeValveR1_OpenStat,
	c1=> ,
	q1=>XV221B_LimeValveR1_CloseCmd ,
	q2=>XV221B_LimeValveR1_OpenCmd );

EQUIP_TYPE_3_Valve3_RB1(
	i1:=NOT reactorB1.q4 OR hold_tertiary_process OR hold_SBR_B,
	i2:= reactorB1.q4,
	s1:= XV211B_AlumValveR1_CloseStat,
	s2:= XV211B_AlumValveR1_OpenStat,
	c1=> ,
	q1=>XV211B_AlumValveR1_CloseCmd ,
	q2=>XV211B_AlumValveR1_OpenCmd );

EQUIP_TYPE_3_Valve4_RB1(
	i1:=NOT reactorB1.q5 OR hold_SBR_B ,
	i2:= reactorB1.q5,
	s1:=XV201B_AirBlowerValveR1_CloseStat ,
	s2:=XV201B_AirBlowerValveR1_OpenStat ,
	c1=> ,
	q1=>XV201B_AirBlowerValveR1_CloseCmd ,
	q2=>XV201B_AirBlowerValveR1_OpenCmd );

EQUIP_TYPE_9_Valve5_RB1(
	i1:= NOT reactorB1.q7 OR hold_SBR_B ,
	i2:=reactorB1.q7 ,
	s1:=XV241B_SludgeValveR1_CloseStat ,
	s2:=XV241B_SludgeValveR1_OpenStat ,
	c1=> ,
	q1=>XV241B_SludgeValveR1_CloseCmd ,
	q2=>XV241B_SludgeValveR1_OpenCmd );

EQUIP_TYPE_10_Dec_RB1(
	i1:=reactorB1.q8 OR NOT hold_SBR_B ,
	i2:= reactorB1.q9 OR NOT hold_SBR_B,
	r1:= reset_dec_RB1,
	s1:= XV261B_DecanterR1_EStopStat,
	s2:= XV261B_DecanterR1_FwdStat,
	s3:= XV261B_DecanterR1_OverloadStat,
	s4:= XV261B_DecanterR1_OverloadStat,
	s5:= XV261B_DecanterR1_RvsStat,
	q1=> XV261B_DecanterR1_RvsCmd,
	q2=>XV261B_DecanterR1_FwdCmd ,
	e1=> );




EQUIP_TYPE_3_Valva1_RB2(
	i1:=NOT reactorB2.q1 OR hold_SBR_B,
	i2:=reactorB2.q1 ,
	s1:=XV206B_SBRValveR2_CloseStat ,
	s2:=XV206B_SBRValveR2_OpenStat ,
	c1=> ,
	q1=>XV206B_SBRValveR2_CloseCmd ,
	q2=>XV206B_SBRValveR2_OpenCmd);

EQUIP_TYPE_8_MIXER_B2(
	i1:= NOT reactorB2.q2 OR hold_SBR_B,
	i2:= reactorB2.q2,
	sa1:=M200B2A_MixerR2_EStopStat,
	sa2:=M200B2A_MixerR2_IncompleteStat ,
	sa3:=M200B2A_MixerR2_LocalRemoteStat ,
	sa4:=M200B2A_MixerR2_OverloadStat ,
	sa5:=M200B2A_MixerR2_RunStat ,
	sb1:=M200B2B_MixerR2_EStopStat,
	sb2:=M200B2B_MixerR2_IncompleteStat ,
	sb3:=M200B2B_MixerR2_LocalRemoteStat ,
	sb4:=M200B2B_MixerR2_OverloadStat ,
	sb5:=M200B2B_MixerR2_RunStat ,
	sc1:=M200B2C_MixerR2_EStopStat,
	sc2:=M200B2C_MixerR2_IncompleteStat ,
	sc3:=M200B2C_MixerR2_LocalRemoteStat ,
	sc4:=M200B2C_MixerR2_OverloadStat ,
	sc5:=M200B2C_MixerR2_RunStat ,
	c1=> ,
	q1=>M200B2A_MixerR2_RunCmd ,
	q2=>M200B2B_MixerR2_RunCmd,
	q3=>M200B2C_MixerR2_RunCmd ,
	e1=> );

EQUIP_TYPE_3_Valve2_RB2(
	i1:=NOT reactorB2.q3 OR hold_SBR_B ,
	i2:= reactorB2.q3,
	s1:= XV222B_LimeValveR2_CloseStat,
	s2:= XV222B_LimeValveR2_OpenStat,
	c1=> ,
	q1=>XV222B_LimeValveR2_CloseCmd ,
	q2=>XV222B_LimeValveR2_OpenCmd );

EQUIP_TYPE_3_Valve3_RB2(
	i1:=NOT reactorB2.q4 OR hold_SBR_B,
	i2:= reactorB2.q4,
	s1:= XV212B_AlumValveR2_CloseStat,
	s2:= XV212B_AlumValveR2_OpenStat,
	c1=> ,
	q1=>XV212B_AlumValveR2_CloseCmd ,
	q2=>XV212B_AlumValveR2_OpenCmd );

EQUIP_TYPE_3_Valve4_RB2(
	i1:=NOT reactorB2.q5 OR hold_SBR_B ,
	i2:= reactorB2.q5,
	s1:=XV202B_AirBlowerValveR2_CloseStat ,
	s2:=XV202B_AirBlowerValveR2_OpenStat ,
	c1=> ,
	q1=>XV202B_AirBlowerValveR2_CloseCmd ,
	q2=>XV202B_AirBlowerValveR2_OpenCmd );


EQUIP_TYPE_9_Valve5_RB2(
	i1:= NOT reactorB2.q7 OR hold_SBR_B ,
	i2:=reactorB2.q7 ,
	s1:=XV242B_SludgeValveR2_CloseStat ,
	s2:=XV242B_SludgeValveR2_OpenStat ,
	c1=> ,
	q1=>XV242B_SludgeValveR2_CloseCmd ,
	q2=>XV242B_SludgeValveR2_OpenCmd );

EQUIP_TYPE_10_Dec_RB2(
	i1:=reactorB2.q8 OR NOT hold_SBR_B ,
	i2:= reactorB2.q9 OR NOT hold_SBR_B,
	r1:= reset_dec_RB2,
	s1:= XV262B_DecanterR2_EStopStat,
	s2:= XV262B_DecanterR2_FwdStat,
	s3:= XV262B_DecanterR2_OverloadStat,
	s4:= XV262B_DecanterR2_OverloadStat,
	s5:= XV262B_DecanterR2_RvsStat,
	q1=> XV262B_DecanterR2_RvsCmd,
	q2=>XV262B_DecanterR2_FwdCmd ,
	e1=> );




EQUIP_TYPE_3_Valva1_RB3(
	i1:=NOT reactorB3.q1 OR hold_SBR_B ,
	i2:=reactorB3.q1 ,
	s1:=XV207B_SBRValveR3_CloseStat ,
	s2:=XV207B_SBRValveR3_OpenStat ,
	c1=> ,
	q1=>XV207B_SBRValveR3_CloseCmd ,
	q2=>XV207B_SBRValveR3_OpenCmd);

EQUIP_TYPE_8_MIXER_B3(
	i1:= NOT reactorB3.q2 OR hold_SBR_B,
	i2:= reactorB3.q2,
	sa1:=M200B3A_MixerR3_EStopStat,
(*	sa2:=M200B3A_MixerR3_IncompleteStat ,*)
	sa3:=M200B3A_MixerR3_LocalRemoteStat ,
	sa4:=M200B3A_MixerR3_OverloadStat ,
	sa5:=M200B3A_MixerR3_RunStat ,
	sb1:=M200B3B_MixerR3_EStopStat,
	sb2:=M200B3B_MixerR3_IncompleteStat ,
	sb3:=M200B3B_MixerR3_LocalRemoteStat ,
	sb4:=M200B3B_MixerR3_OverloadStat ,
	sb5:=M200B3B_MixerR3_RunStat ,
	sc1:=M200B3C_MixerR3_EStopStat,
	sc2:=M200B3C_MixerR3_IncompleteStat ,
	sc3:=M200B3C_MixerR3_LocalRemoteStat ,
	sc4:=M200B3C_MixerR3_OverloadStat ,
	sc5:=M200B3C_MixerR3_RunStat ,
	c1=> ,
	q1=>M200B3A_MixerR3_RunCmd ,
	q2=>M200B3B_MixerR3_RunCmd,
	q3=>M200B3C_MixerR3_RunCmd ,
	e1=> );

EQUIP_TYPE_3_Valve2_RB3(
	i1:=NOT reactorB3.q3 OR hold_SBR_B ,
	i2:= reactorB3.q3,
	s1:= XV223B_LimeValveR3_CloseStat,
	s2:= XV223B_LimeValveR3_OpenStat,
	c1=> ,
	q1=>XV223B_LimeValveR3_CloseCmd ,
	q2=>XV223B_LimeValveR3_OpenCmd );

EQUIP_TYPE_3_Valve3_RB3(
	i1:=NOT reactorB3.q4  OR hold_SBR_B,
	i2:= reactorB3.q4,
	s1:= XV213B_AlumValveR3_CloseStat,
	s2:= XV213B_AlumValveR3_OpenStat,
	c1=> ,
	q1=>XV213B_AlumValveR3_CloseCmd ,
	q2=>XV213B_AlumValveR3_OpenCmd );

EQUIP_TYPE_3_Valve4_RB3(
	i1:=NOT reactorB3.q5 OR hold_SBR_B,
	i2:= reactorB3.q5,
	s1:=XV203B_AirBlowerValveR3_CloseStat ,
	s2:=XV203B_AirBlowerValveR3_OpenStat ,
	c1=> ,
	q1=>XV203B_AirBlowerValveR3_CloseCmd ,
	q2=>XV203B_AirBlowerValveR3_OpenCmd );


EQUIP_TYPE_9_Valve5_RB3(
	i1:= NOT reactorB3.q7  OR hold_SBR_B,
	i2:=reactorB3.q7 ,
	s1:=XV243B_SludgeValveR3_CloseStat ,
	s2:=XV243B_SludgeValveR3_OpenStat ,
	c1=> ,
	q1=>XV243B_SludgeValveClosedR3_CloseCmd ,
	q2=>XV243B_SludgeValveR3_OpenCmd );

EQUIP_TYPE_10_Dec_RB3(
	i1:=reactorB3.q8  OR NOT hold_SBR_B,
	i2:= reactorB3.q9 OR NOT hold_SBR_B,
	r1:= reset_dec_RB3,
	s1:= XV263B_DecanterR3_EStopStat,
	s2:= XV263B_DecanterR3_FwdStat,
	s3:= XV263B_DecanterR3_OverloadStat,
	s4:= XV263B_DecanterR3_OverloadStat,
	s5:= XV263B_DecanterR3_RvsStat,
	q1=> XV263B_DecanterR3_RvsCmd,
	q2=>XV263B_DecanterR3_FwdCmd ,
	e1=> );



EQUIP_TYPE_3_Valva1_RB4(
	i1:=NOT reactorB4.q1 OR hold_SBR_B ,
	i2:=reactorB4.q1 ,
	s1:=XV208B_SBRValveR4_CloseStat ,
	s2:=XV208B_SBRValveR4_OpenStat ,
	c1=> ,
	q1=>XV208B_SBRValveR4_CloseCmd ,
	q2=>XV208B_SBRValveR4_OpenCmd);

EQUIP_TYPE_8_MIXER_B4(
	i1:= NOT reactorB4.q2 OR hold_SBR_B,
	i2:= reactorB4.q2,
	(*sa1:=M200B4A_MixerR4_EStopStat,*)
	sa2:=M200B4A_MixerR4_IncompleteStat ,
	sa3:=M200B4A_MixerR4_LocalRemoteStat ,
	sa4:=M200B4A_MixerR4_OverloadStat ,
	sa5:=M200B4A_MixerR4_RunStat ,
	(*sb1:=M200B4B_MixerR4_EStopStat,*)
	sb2:=M200B4B_MixerR4_IncompleteStat ,
	sb3:=M200B4B_MixerR4_LocalRemoteStat ,
	sb4:=M200B4B_MixerR4_OverloadStat ,
	sb5:=M200B4B_MixerR4_RunStat ,
	(*sc1:=M200B4C_MixerR4_EStopStat,*)
	sc2:=M200B4C_MixerR4_IncompleteStat ,
	sc3:=M200B4C_MixerR4_LocalRemoteStat ,
	sc4:=M200B4C_MixerR4_OverloadStat ,
	sc5:=M200B4C_MixerR4_RunStat ,
	c1=> ,
	q1=>M200B4A_MixerR4_RunCmd ,
	q2=>M200B4B_MixerR4_RunCmd,
	q3=>M200B4C_MixerR4_RunCmd ,
	e1=> );

EQUIP_TYPE_3_Valve2_RB4(
	i1:=NOT reactorB4.q3 OR hold_SBR_B ,
	i2:= reactorB4.q3,
	s1:= XV224B_LimeValveR4_CloseStat,
	s2:= XV224B_LimeValveR4_OpenStat,
	c1=> ,
	q1=>XV224B_LimeValveR4_CloseCmd ,
	q2=>XV224B_LimeValveR4_OpenCmd );

EQUIP_TYPE_3_Valve3_RB4(
	i1:=NOT reactorB4.q4 OR hold_SBR_B ,
	i2:= reactorB4.q4,
	s1:= XV214B_AlumValveR4_CloseStat,
	s2:= XV214B_AlumValveR4_OpenStat,
	c1=> ,
	q1=>XV214B_AlumValveR4_CloseCmd ,
	q2=>XV214B_AlumValveR4_OpenCmd );

EQUIP_TYPE_3_Valve4_RB4(
	i1:=NOT reactorB4.q5 OR hold_SBR_B ,
	i2:= reactorB4.q5,
	s1:=XV204B_AirBlowerValveR4_CloseStat ,
	s2:=XV204B_AirBlowerValveR4_OpenStat ,
	c1=> ,
	q1=>XV204B_AirBlowerValveR4_CloseCmd ,
	q2=>XV204B_AirBlowerValveR4_OpenCmd );

EQUIP_TYPE_9_Valve5_RB4(
	i1:= NOT reactorB4.q7 OR hold_SBR_B ,
	i2:=reactorB4.q7 ,
	s1:=XV244B_SludgeValveR4_CloseStat ,
	s2:=XV244B_SludgeValveR4_OpenStat ,
	c1=> ,
	q1=>XV244B_SludgeValveR4_CloseCmd ,
	q2=>XV244B_SludgeValveR4_OpenCmd );

EQUIP_TYPE_10_Dec_RB4(
	i1:=reactorB4.q8 OR NOT  hold_SBR_B ,
	i2:= reactorB4.q9 OR NOT  hold_SBR_B,
	r1:= reset_dec_RB4,
	s1:= XV264B_DecanterR4_EStopStat,
	s2:= XV264B_DecanterR4_FwdStat,
	s3:= XV264B_DecanterR4_OverloadStat,
	s4:= XV264B_DecanterR4_OverloadStat,
	s5:= XV264B_DecanterR4_RvsStat,
	q1=> XV264B_DecanterR4_RvsCmd,
	q2=>XV264B_DecanterR4_FwdCmd ,
	e1=> );


reset_Pump2_RB := reset_dec_RB1 := reset_dec_RB2 := reset_dec_RB3 := reset_dec_RB4 := RST003B_ResetButtonSBR_2;

timeConversion_alumB1(inputTime:=InputTime_alumB1 , atTime:= alum_reactorB1, outputTime=>OutputTime_alumB1 );
timeConversion_alumB2(inputTime:=InputTime_alumB2 , atTime:= alum_reactorB2, outputTime=>OutputTime_alumB2 );
timeConversion_alumB3(inputTime:=InputTime_alumB3 , atTime:= alum_reactorB3, outputTime=>OutputTime_alumB3 );
timeConversion_alumB4(inputTime:=InputTime_alumB4 , atTime:= alum_reactorB4, outputTime=>OutputTime_alumB4 );
END_ACTION
ACTION reuse_water_FBD:
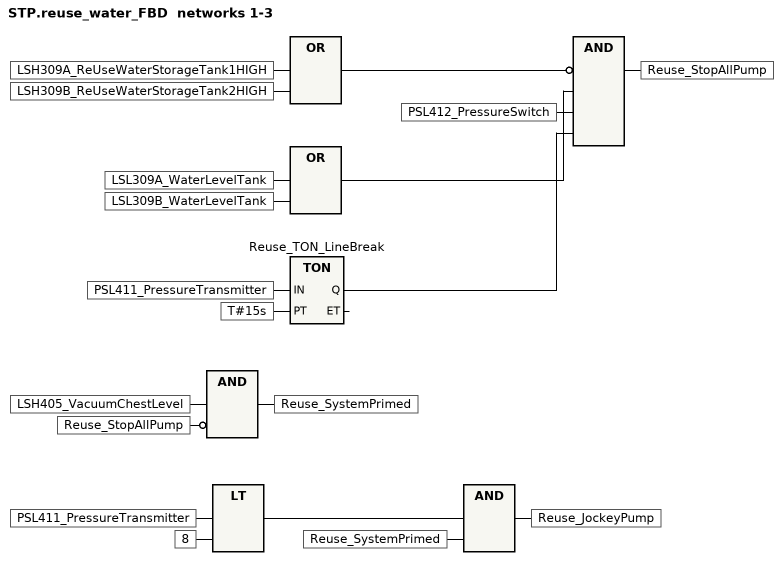
[picture p0: STP.reuse_water_FBD (FBD) networks 1-3]
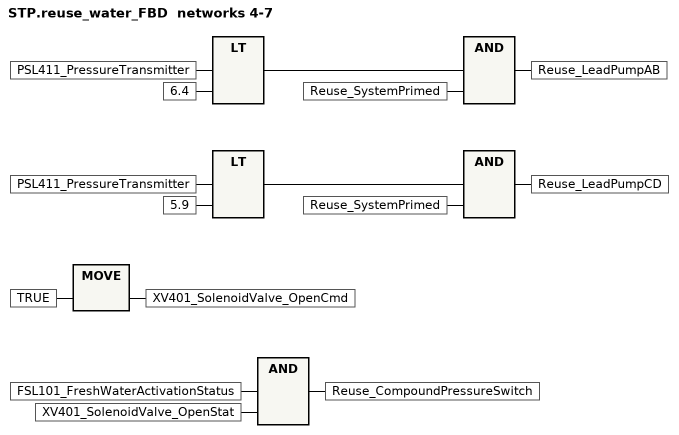
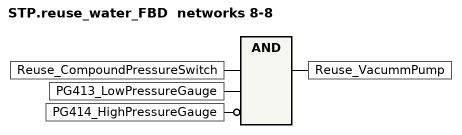
_FBD_ (* Function Block Diagram *)
NETWORK 1
	AND(NOT OR(LSH309A_ReUseWaterStorageTank1HIGH, LSH309B_ReUseWaterStorageTank2HIGH), OR(LSL309A_WaterLevelTank, LSL309B_WaterLevelTank), PSL412_PressureSwitch, Reuse_TON_LineBreak:TON(IN: PSL411_PressureTransmitter, PT: T#15s)) => Reuse_StopAllPump
NETWORK 2
	AND(LSH405_VacuumChestLevel, NOT Reuse_StopAllPump) => Reuse_SystemPrimed
NETWORK 3
	AND(LT(PSL411_PressureTransmitter, 8), Reuse_SystemPrimed) => Reuse_JockeyPump
NETWORK 4
	AND(LT(PSL411_PressureTransmitter, 6.4), Reuse_SystemPrimed) => Reuse_LeadPumpAB
NETWORK 5
	AND(LT(PSL411_PressureTransmitter, 5.9), Reuse_SystemPrimed) => Reuse_LeadPumpCD
NETWORK 6
	MOVE(TRUE) => XV401_SolenoidValve_OpenCmd
NETWORK 7
	AND(FSL101_FreshWaterActivationStatus, XV401_SolenoidValve_OpenStat) => Reuse_CompoundPressureSwitch
NETWORK 8
	AND(Reuse_CompoundPressureSwitch, PG413_LowPressureGauge, NOT PG414_HighPressureGauge) => Reuse_VacummPump
_END_FBD_
(* the same logic as Structured Text *)
(* Network 1 *)
Reuse_TON_LineBreak(IN := PSL411_PressureTransmitter, PT := T#15s);
Reuse_StopAllPump := NOT (LSH309A_ReUseWaterStorageTank1HIGH OR LSH309B_ReUseWaterStorageTank2HIGH) AND (LSL309A_WaterLevelTank OR LSL309B_WaterLevelTank) AND PSL412_PressureSwitch AND Reuse_TON_LineBreak.Q;
(* Network 2 *)
Reuse_SystemPrimed := LSH405_VacuumChestLevel AND NOT Reuse_StopAllPump;
(* Network 3 *)
Reuse_JockeyPump := (PSL411_PressureTransmitter < 8) AND Reuse_SystemPrimed;
(* Network 4 *)
Reuse_LeadPumpAB := (PSL411_PressureTransmitter < 6.4) AND Reuse_SystemPrimed;
(* Network 5 *)
Reuse_LeadPumpCD := (PSL411_PressureTransmitter < 5.9) AND Reuse_SystemPrimed;
(* Network 6 *)
XV401_SolenoidValve_OpenCmd := TRUE;
(* Network 7 *)
Reuse_CompoundPressureSwitch := FSL101_FreshWaterActivationStatus AND XV401_SolenoidValve_OpenStat;
(* Network 8 *)
Reuse_VacummPump := Reuse_CompoundPressureSwitch AND PG413_LowPressureGauge AND NOT PG414_HighPressureGauge;
END_ACTION
ACTION reuse_water_ST:
(*
REUSE_WATER_A(
	i3:= PSL412_PressureSwitch,
	i1:= LSL309A_WaterLevelTank,
	i4:= LSH405_VacuumChestLevel,
	i2:= (*unused*),
	i5:= PG413_LowPressureGauge,
	i6:= PG414_HighPressureGauge,
	p1:= PSL411_PressureTransmitter,
	q1=> ,
	q2=> ,
	q3=> ,
	q4=> ,
	q5=> ,
	q6=> ,
	q7=> ,
	q8=> ,
	q9=> );
*)

EQUIP_TYPE_2_P402(
	i1:=REUSE_WATER_A.q1 OR hold_reuse_process,
	i2:=REUSE_WATER_A.q2 ,
	sa1:= P402A_JockeyPumpA_EStopStat ,
	sa2:= P402A_JockeyPumpA_IncompleteStat,
	sa3:= P402A_JockeyPumpA_LocalRemoteStat,
	sa4:= P402A_JockeyPumpA_OverloadStat,
	sa5:= P402A_JockeyPumpA_OnOffStat,
	sb1:= P402B_JockeyPumpB_EStopStat,
	sb2:= P402B_JockeyPumpB_IncompleteStat,
	sb3:= P402B_JockeyPumpB_LocalRemoteStat,
	sb4:= P402B_JockeyPumpB_OverloadStat,
	sb5:= P402B_JockeyPumpB_OnOffStat,
	c1=> ,
	q1=> P402A_JockeyPumpA_RunCmd,
	q2=> P402B_JockeyPumpB_RunCmd ,
	e1=> );

EQUIP_TYPE_2_P401AB(
	i1:=REUSE_WATER_A.q3 OR hold_reuse_process ,
	i2:=REUSE_WATER_A.q4 ,
	sa1:= P401A_LeadPumpA_EStopStat,
	sa2:= P401A_LeadPumpA_IncompleteStat,
	sa3:= P401A_LeadPumpA_LocalRemoteStat,
	sa4:= P401A_LeadPumpA_OverloadStat,
	sa5:= P401A_LeadPumpA_OnOffStat,
	sb1:= P401B_LeadPumpB_EStopStat,
	sb2:= P401B_LeadPumpB_IncompleteStat,
	sb3:= P401B_LeadPumpB_LocalRemoteStat,
	sb4:= P401B_LeadPumpB_OnOffStat,
	sb5:= P401B_LeadPumpB_OverloadStat,
	c1=> ,
	q1=> P401A_LeadPumpA_RunCmd,
	q2=> P401B_LeadPumpB_RunCmd,
	e1=> );

EQUIP_TYPE_2_P401CD(
	i1:= REUSE_WATER_A.q5 OR hold_reuse_process,
	i2:= REUSE_WATER_A.q6,
	sa1:= P401C_LeadPumpC_EStopStat,
	sa2:= P401C_LeadPumpC_IncompleteStat,
	sa3:= P401C_LeadPumpC_LocalRemoteStat,
	sa4:= P401C_LeadPumpC_OverloadStat,
	sa5:= P401C_LeadPumpC_OnOffStat,
	sb1:= P401D_LeadPumpD_EStopStat,
	sb2:= P401D_LeadPumpD_IncompleteStat,
	sb3:= P401D_LeadPumpD_LocalRemoteStat,
	sb4:= P401D_LeadPumpD_OverloadStat,
	sb5:= P401D_LeadPumpD_OnOffStat,
	c1=> ,
	q1=> P401C_LeadPumpC_RunCmd,
	q2=> P401D_LeadPumpD_RunCmd,
	e1=> );

EQUIP_TYPE_2_P403(
	i1:=REUSE_WATER_A.q7 OR hold_reuse_process ,
	i2:=REUSE_WATER_A.q8 ,
	sa1:= P403A_VacuumPumpA_EStopStat ,
	sa2:= ,
	sa3:= P403A_VacuumPumpA_LocalRemoteStat,
	sa4:= P403A_VacuumPumpA_OverloadStat,
	sa5:= P403A_VacuumPumpA_OnOffStat,
	sb1:= P403B_VacuumPumpB_EStopStat,
	sb2:= ,
	sb3:= P403B_VacuumPumpB_LocalRemoteStat,
	sb4:= P403B_VacuumPumpB_OverloadStat,
	sb5:= P403B_VacuumPumpB_OnOffStat,
	c1=> ,
	q1=> P403A_VacuumPumpA_RunCmd,
	q2=> P403B_VacuumPumpB_RunCmd,
	e1=> );

EQUIP_TYPE_5_xv401(
	i1:= NOT REUSE_WATER_A.q9 OR hold_reuse_process,
	i2:= REUSE_WATER_A.q9 ,
	sa1:=XV401_SolenoidValve_CloseStat ,
	sa2:=XV401_SolenoidValve_OpenStat ,
	c1=> ,
	q1=> XV401_SolenoidValve_OpenCmd,
	e1=> );

IF  GenActive THEN
P401A_LeadPumpA_RunCmd := FALSE;
P401B_LeadPumpB_RunCmd := FALSE;
P401C_LeadPumpC_RunCmd := FALSE;
P401D_LeadPumpD_RunCmd := FALSE;
END_IF
END_ACTION
ACTION tertiary:
IF NOT hold_tertiary_process THEN
tertiary_treatment_plant_A(
	i1:= LSH301_EffluentSump,
	i2:= LSL309A_WaterLevelTank,
	i3:= LSL301_EffluentSump,
	i4:= LSH301_EffluentSump,
	i5:= LSH302_CollectionSump,
	i6:= LSH501A_SludgeStorage AND LSH501B_SludgeStorage,
	i7:= LSHH501A_SludgeStorage AND LSHH501B_SludgeStorage,
	s1:= K301A_AirCompressor_RunStat,
	s2:= K301B_AirCompressor_RunStat,
	s3:= P301A_EffluentTransferPump_RunStat,
	s4:= P301B_EffluentTransferPump_RunStat ,
	q1=> , 
	q2=> , 
	q3=> , 
	q4=> ,
	q5=> ,
	q6=> ,
	q7=> ,
	q8=> ,
	q9=> ,
	q10=> , 
	q11=> ,
	q12=> );
END_IF

EQUP_TYPE_1_P301(
	i1:= tertiary_treatment_plant_A.q1 OR hold_tertiary_process,
	i2:= tertiary_treatment_plant_A.q2,
	r1:=reset_tertiary_p301 ,
	sa1:= P301A_EffluentTransferPump_EStopStat,
	sa2:= ,
	sa3:= P301A_EffluentTransferPump_LocalRemoteStat,
	sa4:= P301A_EffluentTransferPump_TripStat,
	sa5:= P301A_EffluentTransferPump_RunStat,
	sb1:= P301B_EffluentTransferPump_EStopStat,
	sb2:= ,
	sb3:= P301B_EffluentTransferPump_LocalRemoteStat,
	sb4:= P301B_EffluentTransferPump_TripStat,
	sb5:= P301B_EffluentTransferPump_RunStat,
	c1=> ,
	c2=> ,
	q1=> P301A_EffluentTransferPump_RunCmd,
	q2=> P301B_EffluentTransferPump_RunCmd,
	e1=> );

EQUIP_TYPE_4_M303A(
	i1:= tertiary_treatment_plant_A.q3 OR hold_tertiary_process,
	i2:=tertiary_treatment_plant_A.q4 ,
	sa1:= ,
	sa2:= ,
	sa3:= M303A_Floculator_TripStat,
	sa4:= M303A_Floculator_RunStat,
	c1=> ,
	q1=> M303A_Floculator_RunCmd,
	e1=> );

EQUIP_TYPE_4_M303B(
	i1:= tertiary_treatment_plant_A.q3 OR hold_tertiary_process,
	i2:=tertiary_treatment_plant_A.q4 ,
	sa1:= ,
	sa2:= ,
	sa3:= M303B_Floculator_TripStat,
	sa4:= M303B_Floculator_RunStat,
	c1=> ,
	q1=> M303B_Floculator_RunCmd,
	e1=> );

EQUIP_TYPE_4_M303C(
	i1:= tertiary_treatment_plant_A.q3 OR hold_tertiary_process,
	i2:=tertiary_treatment_plant_A.q4 ,
	sa1:= ,
	sa2:= ,
	sa3:= M303C_Floculator_TripStat,
	sa4:= M303C_Floculator_RunStat,
	c1=> ,
	q1=> M303C_Floculator_RunCmd,
	e1=> );

EQUP_TYPE_1_K301(
	i1:= tertiary_treatment_plant_A.q5 OR hold_tertiary_process,
	i2:= tertiary_treatment_plant_A.q6,
	r1:= reset_tertiary_k301,
	sa1:= K301A_AirCompressor_EStopStat,
	sa2:= ,
	sa3:= K301A_AirCompressor_LocalRemoteStat,
	sa4:= K301A_AirCompressor_TripStat,
	sa5:= K301A_AirCompressor_RunStat,
	sb1:= K301B_AirCompressor_EStopStat,
	sb2:= ,
	sb3:= K301B_AirCompressor_LocalRemoteStat,
	sb4:= K301B_AirCompressor_TripStat,
	sb5:= K301B_AirCompressor_RunStat ,
	c1=> ,
	c2=> ,
	q1=> ,
	q2=> ,
	e1=> );

EQUIP_TYPE_5_XV305(
	i1:=tertiary_treatment_plant_A.q7 OR hold_tertiary_process ,
	i2:=tertiary_treatment_plant_A.q8 ,
	sa1:= XV305_TertiaryTreatmentMainValve_CloseStat,
	sa2:= XV305_TertiaryTreatmentMainValve_OpenStat,
	c1=> ,
	q1=> XV305_TertiaryTreatmentMainValve_OpenCmd,
	e1=> );

EQUP_TYPE_1_p302(
	i1:= tertiary_treatment_plant_A.q9 OR hold_tertiary_process,
	i2:= tertiary_treatment_plant_A.q10,
	r1:= reset_tertiary_p302,
	sa1:= P302A_CollectionPump_EStopStat,
	sa2:= ,
	sa3:= P302A_CollectionPump_LocalRemoteStat,
	sa4:= P302A_CollectionPump_TripStat,
	sa5:= P302A_CollectionPump_RunStat,
	sb1:= P302B_CollectionPump_EStopStat,
	sb2:= ,
	sb3:= P302B_CollectionPump_LocalRemoteStat,
	sb4:= P302B_CollectionPump_TripStat,
	sb5:= P302B_CollectionPump_RunStat,
	c1=> ,
	c2=> ,
	q1=> ,
	q2=> ,
	e1=> );

EQUIP_TYPE_5_XV303A(
	i1:= tertiary_treatment_plant_A.q11 OR hold_tertiary_process,
	i2:= tertiary_treatment_plant_A.q12,
	sa1:= XV303A_LamellaSludgeDischarge_CloseStat,
	sa2:= XV303A_LamellaSludgeDischarge_OpenStat,
	c1=> ,
	q1=> XV303A_LamellaSludgeDischarge_RunCmd,
	e1=> );

EQUIP_TYPE_5_XV303B(
	i1:= tertiary_treatment_plant_A.q11 OR hold_tertiary_process,
	i2:= tertiary_treatment_plant_A.q12,
	sa1:= XV303B_LamellaSludgeDischarge_CloseStat,
	sa2:= XV303B_LamellaSludgeDischarge_OpenStat,
	c1=> ,
	q1=> XV303B_LamellaSludgeDischarge_RunCmd,
	e1=> );


EQUIP_TYPE_5_XV303C(
	i1:= tertiary_treatment_plant_A.q11 OR hold_tertiary_process,
	i2:= tertiary_treatment_plant_A.q12,
	sa1:= XV303C_LamellaSludgeDischarge_CloseStat,
	sa2:= XV303C_LamellaSludgeDischarge_OpenStat,
	c1=> ,
	q1=> XV303C_LamellaSludgeDischarge_RunCmd,
	e1=> );


EQUIP_TYPE_5_XV303D(
	i1:= tertiary_treatment_plant_A.q11 OR hold_tertiary_process,
	i2:= tertiary_treatment_plant_A.q12,
	sa1:= XV303D_LamellaSludgeDischarge_CloseStat,
	sa2:= XV303D_LamellaSludgeDischarge_OpenStat,
	c1=> ,
	q1=> XV303D_LamellaSludgeDischarge_RunCmd,
	e1=> );


reset_tertiary_p301 := reset_tertiary_k301 := reset_tertiary_p302 := RST004_ResetButtonChemicalTertiary ;
END_ACTION

(* POU INLET, ST *)
FUNCTION_BLOCK INLET
VAR_INPUT
(*inlet*)
	i1: BOOL;
	i3: BOOL;
	i2: BOOL;
	i4: BOOL;

(*MIXER*)

	i5: BOOL;
	i6: BOOL;

(*penstock*)
	r1: BOOL; (*rs1*)
	i7: BOOL; (*ps open*)
	i8: BOOL;	(*ps open*)
	i10: BOOL;
	i9: BOOL;
	i11: BOOL;
	s1: BOOL;
	s2: BOOL;
	s3: BOOL;
	s4: BOOL;

(* sbr transfer *)
	i12: BOOL;
	i13: BOOL;
	i14: BOOL;
END_VAR
VAR_OUTPUT

(*inlet*)
	q1: BOOL;
	q2: BOOL;

(*MIXER*)

	q3: BOOL;
	q4: BOOL;

(*penstock*)
	q5: BOOL; (*ps1*)
	q6: BOOL; (*ps2*)
	q7: BOOL;
	q8: BOOL;
	q10: BOOL;
	q9: BOOL;
	q11: BOOL;
	q12: BOOL;
	q13: BOOL;
	q14: BOOL;
	q15: BOOL;
	q16: BOOL;
	q17: BOOL;
	q18: BOOL;
	q19: BOOL;
	q20: BOOL;
(* Grit Removal*)

	q21: BOOL;
	q22: BOOL;
	q23: BOOL;
	q24: BOOL;
	q25:BOOL;
	q26:BOOL;

(* sbr transfer *)

	q27: BOOL;
	q28: BOOL;

END_VAR
VAR
(*inlet*)
	m1: BOOL;
	ton1: TON;

(*MIXER*)


(*penstock*)
	penstock: INT;
	FailedGroupA: BOOL;
	FailedGroupB: BOOL;
	m2: BOOL;
	TP1: TP;
	m3: BOOL;
	TON2: TON;
	TON3: TON;
	TOF1: TOF;
	TON4 : TON;
	mr: BOOL;
	F_TRIG1: F_TRIG;
	R_TRIG1: R_TRIG;
	m4 : BOOL;
	TON5: TON;

END_VAR



(*
CASE penstock OF
0:
	q5 := TRUE;
	q6 := FALSE;
	IF FailedGroupA OR m2 THEN
		penstock := 1;
	END_IF
1 :
 	q6 := TRUE;
	IF FailedGroupB THEN
		penstock := 2;
	ELSIF i8 THEN
		penstock := 3;
	END_IF
2 :
	q5 := FALSE;
	q6 := FALSE;
	IF r1 THEN
		penstock := 0;
	END_IF
3:
	q6 := TRUE;
	q5 := FALSE;
	IF FailedGroupB OR m2 THEN
		penstock := 4;
	END_IF
4 :
	q6 := TRUE;
	IF FailedGroupA THEN
		penstock := 2;
	ELSIF i7 THEN
		penstock := 0;
	END_IF
END_CASE*)
(*EQ Pump*)
q1 := NOT i1 OR i3 OR m1;
q2 := i2 AND NOT i3 AND NOT m1;
ton1(IN:=i4 , PT:=t#5m , Q=>m1 , ET=> );

(*Mixer*)
q3 := NOT i5;
q4 := i6;


(*screen*)
FailedGroupA := s1 OR s2;
FailedGroupB := s3 OR s4;

m4 := ((NOT m4 AND (FailedGroupA OR m2)) OR m4) AND NOT((m4 AND (FailedGroupB OR m2)) OR r1);
q5 := (NOT m4 OR q5) AND NOT(( m4 AND i8) OR mr) ;
q6 := (m4 OR q6) AND NOT ((NOT m4 AND i7) OR mr);
mr := (mr OR (FailedGroupA AND FailedGroupB)) AND NOT r1;

TOF1(IN:=i11 , PT:=T#2m , Q=>i9 , ET=> );

(*rectifuy using reset button*)
F_TRIG1(CLK:=m4 );
R_TRIG1(CLK:=m4 );
TP1(IN:=(F_TRIG1.Q OR R_TRIG1.Q) , PT:= T#5m , Q=>m3 , ET=> );
m2 := i10 AND NOT m3;

TON4(IN:=NOT i9 OR NOT(q5 OR q6) , PT:=T#5m , Q=>q7 , ET=> );
TON2(IN:= i9 AND (q5 OR q6), PT := T#1h, Q=> q8);

TON3(IN:=q7,PT:=T#5m,Q=>q9);
q10 := q8;

q11 := q9;
q12 := q10;

q13 := NOT (i9 AND Q5);
q14 := (i9 AND Q5);

q15 := NOT(i9 AND q6);
q16 := (i9 AND q6);

q17 := q13;
q18 := q14;

q19 := q15;
q20 :=q18;

(*Grit Removal*)
q21 := i7;
q22 := i8;

q23 := NOT i9;
q24 := i9;

TON5(IN:= NOT i9, PT:=T#5m , Q=>q25 );
q26 := i9;


(*sbr transfer*)
q27  := (NOT i12) OR NOT i14;
q28 := i13 AND i14;
END_FUNCTION_BLOCK

(* POU EQUIP_TYPE_1, ST *)
FUNCTION_BLOCK EQUIP_TYPE_1
VAR_INPUT
	i1 : BOOL;
	i2 : BOOL;
	r1 : BOOL;

	sa1 : BOOL;
	sa2 : BOOL;
	sa3 : BOOL;
	sa4 : BOOL;
	sa5 : BOOL;

	sb1 : BOOL;
	sb2 : BOOL;
	sb3 : BOOL;
	sb4 : BOOL;
	sb5 : BOOL;
END_VAR
VAR_OUTPUT
	c1 : BOOL;
	c2 :BOOL;
	q1 : BOOL;
	q2 : BOOL;
	e1 : BOOL;
END_VAR
VAR
	toggle : INT;
END_VAR
c1 := (i2 OR c1) AND NOT i1;
e1 :=(( (sa2 OR sa4 OR sa1) AND (sb2 OR sb4 OR sb1)) OR e1) AND NOT r1;

CASE toggle OF
0:
	c2 := TRUE;
	IF e1 THEN
		toggle := 3;
	ELSIF sa2 OR sa4 OR sa1 THEN
		toggle := 1;
	END_IF
1:
	c2 := FALSE;
	IF e1 THEN
		toggle := 3;
	ELSIF  sb2 OR sb4 OR sb1  THEN
		toggle := 0;
	END_IF
3:
	IF r1 THEN
		toggle := 0;
	END_IF

END_CASE

q1 := c1 AND NOT c2 AND NOT(sa1 OR sa3 );
q2 := c1 AND c2 AND NOT(sb1 OR sb3 );


IF phaselock THEN
q1:=FALSE;
q2:=FALSE;
END_IF
END_FUNCTION_BLOCK

(* POU EQUIP_TYPE_2, ST *)
FUNCTION_BLOCK EQUIP_TYPE_2 (*dual equipment*)
VAR_INPUT
	i1 : BOOL;
	i2 : BOOL;

	sa1 : BOOL;
	sa2 : BOOL;
	sa3 : BOOL;
	sa4 : BOOL;
	sa5 : BOOL;

	sb1 : BOOL;
	sb2 : BOOL;
	sb3 : BOOL;
	sb4 : BOOL;
	sb5 : BOOL;
END_VAR
VAR_OUTPUT
	c1 : BOOL;
	q1 : BOOL;
	q2 : BOOL;
	e1 : BOOL;
END_VAR
VAR
END_VAR
c1 := (i2 OR c1) AND NOT i1;
e1 :=(( (sa2 OR sa4 OR sa1 OR sa3) AND (sb2 OR sb4 OR sb1  OR sa3)));
q1 := c1 AND NOT (sa2 OR sa4 OR sa1 OR sa3) ;
q2 := c1 AND NOT (sb2 OR sb4 OR sb1  OR sa3) ;


IF phaselock THEN
q1:=FALSE;
q2:=FALSE;
END_IF
END_FUNCTION_BLOCK

(* POU EQUIP_TYPE_3, ST *)
FUNCTION_BLOCK EQUIP_TYPE_3 (*penstock*)
VAR_INPUT
	i1:BOOL;
	i2 : BOOL;
	s1:BOOL;
	s2:BOOL;
	s3:BOOL;
	s4:BOOL;
END_VAR
VAR_OUTPUT
	c1 : BOOL;
	q1: BOOL;
	q2: BOOL;
END_VAR
VAR
END_VAR
c1 := (i2 OR c1) AND NOT( i1 OR s2 OR s4);
q1 := NOT c1;
q2 := c1;


IF phaselock THEN
q1:=FALSE;
q2:=FALSE;
END_IF
END_FUNCTION_BLOCK

(* POU EQUIP_TYPE_4, ST *)
FUNCTION_BLOCK EQUIP_TYPE_4
(*
	single equipment
	sa1:= F101B2_FineScr_EStopStat,
	sa2:= F101B2_FineScr_LocalRemoteStat,
	sa3:= F101B2_FineScr_OverloadStat,
	sa4:= F101B2_FineScr_RunStat,
*)
VAR_INPUT
	i1 : BOOL;
	i2 : BOOL;

	sa1 : BOOL;
	sa2 : BOOL;
	sa3 : BOOL;
	sa4 : BOOL;

END_VAR
VAR_OUTPUT
	c1 : BOOL;
	q1 : BOOL;
	e1 : BOOL;
END_VAR
VAR
END_VAR
c1 := (i2 OR c1) AND NOT i1;
e1 :=( ( sa3 OR sa1));
q1 := c1 AND NOT (e1 OR sa2);


IF phaselock THEN
q1:=FALSE;
END_IF
END_FUNCTION_BLOCK

(* POU EQUIP_TYPE_5, ST *)
FUNCTION_BLOCK EQUIP_TYPE_5 (*general valve*)
VAR_INPUT
	i1 : BOOL;
	i2 : BOOL;

	sa1 : BOOL;
	sa2 : BOOL;

END_VAR
VAR_OUTPUT
	c1 : BOOL;
	q1 : BOOL;
	e1 : BOOL;
END_VAR
VAR
END_VAR
c1 := (i2 OR c1) AND NOT i1;
q1 := c1;


IF phaselock THEN
q1:=FALSE;
END_IF
END_FUNCTION_BLOCK

(* POU EQUIP_TYPE_6, ST *)
FUNCTION_BLOCK EQUIP_TYPE_6 (*Valve with TIMER*)
VAR_INPUT
	i1 : BOOL;
	i2 : BOOL;

	sa1 : BOOL;
	sa2 : BOOL;

END_VAR
VAR_OUTPUT
	c1 : BOOL;
	q1 : BOOL;
	e1 : BOOL;
END_VAR
VAR
	TON1: TON;
	TON2: TON;
END_VAR
c1 := (i2 OR c1) AND NOT i1;
TON1(IN:= NOT TON2.Q AND c1, PT:= T#1m, Q=> , ET=> );
TON2(IN:=TON1.Q , PT:= T#5m, Q=> , ET=> );
q1 := (NOT TON1.Q) AND c1 ;


IF phaselock THEN
q1:=FALSE;
END_IF
END_FUNCTION_BLOCK

(* POU EQUIP_TYPE_7, ST *)
FUNCTION_BLOCK EQUIP_TYPE_7 (* cycle done *)
VAR_INPUT
	i1 : BOOL;
	i2 : BOOL;
	r1 : BOOL;

	sa1 : BOOL;
	sa2 : BOOL;
	sa3 : BOOL;
	sa4 : BOOL;
	sa5 : BOOL;

	sb1 : BOOL;
	sb2 : BOOL;
	sb3 : BOOL;
	sb4 : BOOL;
	sb5 : BOOL;
END_VAR
VAR_OUTPUT
	c1 : BOOL;
	c2 :BOOL;
	q1 : BOOL;
	q2 : BOOL;
	e1 : BOOL;
END_VAR
VAR
	toggle : INT;
	TON1: TON;
END_VAR
c1 := (i2 OR c1) AND NOT i1;
e1 :=(( (sa2 OR sa4 OR sa1) AND (sb2 OR sb4 OR sb1)) OR e1) AND NOT r1;

CASE toggle OF
0:
	c2 := TRUE;
	TON1(IN:=TRUE , PT:= T#2h, Q=> , ET=> );
	IF e1 THEN
		toggle := 3;
		TON1(IN:=FALSE , PT:= T#2h, Q=> , ET=> );
	ELSIF sa2 OR sa4 OR sa1 OR TON1.Q THEN
		toggle := 1;
		TON1(IN:=FALSE , PT:= T#2h, Q=> , ET=> );
	END_IF
1:
	c2 := FALSE;
	TON1(IN:=TRUE , PT:= T#2h, Q=> , ET=> );
	IF e1 THEN
		toggle := 3;
		TON1(IN:=FALSE , PT:= T#2h, Q=> , ET=> );
	ELSIF  sb2 OR sb4 OR sb1 OR TON1.Q THEN
		toggle := 0;
		TON1(IN:=FALSE , PT:= T#2h, Q=> , ET=> );
	END_IF
3:
	IF r1 THEN
		toggle := 0;
	END_IF

END_CASE

q1 := c1 AND NOT c2 AND NOT(sa3);
q2 := c1 AND c2 AND NOT(sb3);


IF phaselock THEN
q1:=FALSE;
q2:=FALSE;
END_IF
END_FUNCTION_BLOCK

(* POU Chemical_new, ST *)
FUNCTION_BLOCK Chemical_new
VAR_INPUT
	iA1: BOOL;
	iA2: BOOL;
	iA3: BOOL;
	iA4: BOOL;
	rA1: BOOL;

	iB1: BOOL;
	iB2: BOOL;
	iB3: BOOL;
	iB4: BOOL;
	rB1: BOOL;

	iC1: BOOL;
	iC2: BOOL;
	iC3: BOOL;
	iC4: BOOL;
	rC1: BOOL;


	iqA2: BOOL;
	iqB2: BOOL;
	iqC2: BOOL;


	iLRA: BOOL;
	iLRB: BOOL;

	iAop1: BOOL;
	iAop2: BOOL;
	iAop3: BOOL;
	iAop4: BOOL;



	iAlss1: BOOL;
	iAlss2: BOOL;
	iAlss3: BOOL;
	iAlss4: BOOL;

	iasbrA: BOOL; (*sbr alum vale*)
	iasbrB: BOOL;

	iCop1 : BOOL;
	iCop2 : BOOL;
	ilssC1 : BOOL;
	ilssC2 : BOOL;

	itpm : BOOL;

	ilssch1: BOOL;
	ilssch2: BOOL;
	ilssch3: BOOL;

	iChop1: BOOL;
	iChop2: BOOL;
	iChop3: BOOL;

	irdAB : BOOL;

	PHT301: REAL;
	CL303: REAL;

END_VAR
VAR_OUTPUT
	qA1: BOOL;
	qA2: BOOL;
	qA3: BOOL;
	eA1: BOOL;

	qB1: BOOL;
	qB2: BOOL;
	qB3: BOOL;
	eB1: BOOL;

	qC1: BOOL;
	qC2: BOOL;
	qC3: BOOL;
	eC1: BOOL;

	qD1: BOOL;
	qD2: BOOL;
	qD3: BOOL;
	eD1: BOOL;

	qCir: BOOL;

	qLA: BOOL;
	qLB: BOOL;

	qP1: BOOL;
	qP2: BOOL;

	qP3: BOOL;
	qP4: BOOL;

	qtA1: BOOL;
	qtC1: BOOL;
	qtCH1: BOOL;

	qdsp : BOOL;


END_VAR
VAR
	tank_lime_A: tanks;
	tank_lime_B: tanks;
	tank_lime_C: tanks;


	alumtankstat: BOOL;
	limetankstat: BOOL;
	caustictankstat: BOOL;
	chlorintankstat: BOOL;

	causticDosing: BOOL;
	chlorinDosing: BOOL;
END_VAR
tank_lime_A(
	LSLL:=iA1 ,
	LSL:= iA2,
	LSH:= iA3,
	LSHH:=iA4 ,
	reset:= rA1,
	fill=> qA1,
	valve=> qA2,
	mixer=> qA3,
	alarm=>eA1 );

tank_lime_B(
	LSLL:=iB1 ,
	LSL:= iB2,
	LSH:= iB3,
	LSHH:=iB4 ,
	reset:= rB1,
	fill=> qB1,
	valve=> qB2,
	mixer=> qB3,
	alarm=>eB1 );

tank_lime_C(
	LSLL:=iC1 ,
	LSL:= iC2,
	LSH:= iC3,
	LSHH:=iC4 ,
	reset:= rC1,
	fill=> qC1,
	valve=> qC2,
	mixer=> qC3,
	alarm=>eC1 );


qCir := TRUE;

qLA := iLRA;
qLB := iLRB;

limetankstat;


qP1 :=iLRA AND (iqA2 OR iqB2 OR iqC2);
qP2 := iLRA AND (iqA2 OR iqB2 OR iqC2);

alumtankstat := (iAlss1 AND iAop1) OR (iAlss2 AND iAop2) OR (iAlss3 AND iAop3) OR (iAlss4 AND iAop4);

(*Alum tank*)
qP3 := iasbrA AND alumtankstat;
qP4 := iasbrB AND alumtankstat;

(*alum tank tertiary*)
qtA1 := itpm AND alumtankstat;


(*caustic*)
caustictankstat := (ilssc1 AND iCop1) OR (ilssc2 AND iCop2);

qtC1 := caustictankstat AND itpm AND causticDosing ; (*ph value*)



(*clorin*)
chlorintankstat := (ilssch1 AND iChop1) OR (ilssch2 AND iChop2) OR (ilssch3 AND iChop3);
chlorinDosing := (chlorinDosing OR CL303 < 6.5) AND NOT (CL303 > 7);
qtCH1 := chlorintankstat AND itpm AND chlorinDosing;

(*effuent disinfection*)
qdsp := irdAB AND chlorintankstat;
END_FUNCTION_BLOCK

(* POU tanks, ST *)
FUNCTION_BLOCK tanks
VAR_INPUT
	LSLL: BOOL;
	LSL: BOOL;
	LSH: BOOL;
	LSHH: BOOL;

	reset: BOOL;

END_VAR
VAR_OUTPUT

	fill: BOOL;
	valve: BOOL;
	mixer: BOOL;
	alarm: BOOL;
END_VAR
VAR
	tank: INT;
END_VAR
IF NOT  LSLL THEN
	fill := TRUE;
ELSIF LSHH THEN
	fill:= FALSE;
END_IF

valve := FALSE;
alarm := FALSE;
CASE tank OF
0: IF lsh THEN
	tank := 1;
	alarm := TRUE;
      END_IF
1:
	IF reset THEN
		alarm := FALSE;
		valve := TRUE;
		tank := 2;
	END_IF
2 :
	IF NOT lsll THEN
		tank := 0;
	END_IF
END_CASE

IF LSH THEN
	mixer := TRUE;
ELSIF NOT LSL THEN
	mixer := FALSE;
END_IF
END_FUNCTION_BLOCK

(* POU EQUIPMENT_REDUNDANT_AIRBLOWER, ST *)
FUNCTION_BLOCK EQUIPMENT_REDUNDANT_AIRBLOWER
VAR_INPUT
	i1 : BOOL;
	i2 : BOOL;
	i3 : BOOL;
	i4 : BOOL;

	sa1 : BOOL;
	sa2 : BOOL;
	sa3 : BOOL;
	sa4 : BOOL;
	sa5 : BOOL;

	sb1 : BOOL;
	sb2 : BOOL;
	sb3 : BOOL;
	sb4 : BOOL;
	sb5 : BOOL;

	sc1 : BOOL;
	sc2 : BOOL;
	sc3 : BOOL;
	sc4 : BOOL;
	sc5 : BOOL;

	r1: BOOL;

END_VAR
VAR_OUTPUT
	q1 : BOOL;
	q2 : BOOL;
	q3 : BOOL;
	e1: BOOL;
END_VAR
VAR
	c1 : BOOL;
	c2 : BOOL;
	c3: BOOL;
END_VAR
(*

EQUIPMENT_REDUNDANT_AIRBLOWER_2_Sludge1(
	i1:= sludge_holding_A.q1A,
	i2:= sludge_holding_A.q2A,
	i3:= sludge_holding_A.q1B,
	i4:= sludge_holding_A.q2B,
	sa1:=B501A_Blower_EStopStat ,
	sa2:= B501A_Blower_IncompleteStat,
	sa3:= B501A_Blower_LocalRemoteStat,
	sa4:= B501A_Blower_OverloadStat,
	sa5:= B501A_Blower_RunStat,
	sb1:= B501B_Blower_EStopStat,
	sb2:= B501B_Blower_IncompleteStat,
	sb3:= B501B_Blower_LocalRemoteStat,
	sb4:= B501B_Blower_OverloadStat,
	sb5:= B501B_Blower_RunStat,
	sc1:= B501C_Blower_EStopStat,
	sc2:= B501C_Blower_IncompleteStat,
	sc3:= B501C_Blower_LocalRemoteStat,
	sc4:= B501C_Blower_OverloadStat,
	sc5:= B501C_Blower_RunStat,
	q1=> B501A_Blower_RunCmd,
	q2=> B501B_Blower_RunCmd,
	q3=> B501C_Blower_RunCmd);

*)

c1 :=  (i2 OR c1) AND ( i1 OR (sa1 OR sa2 OR sa4 OR NOT sa3)) ;
c2 :=  (i4 OR c2) AND ( i3 OR  (sb1 OR sb2 OR sb4 OR NOT sb3));


IF r1 THEN
	e1 := FALSE;
ELSIF e1 THEN
	c1 := FALSE;
	c2 := FALSE;
	c3 := FALSE;
ELSIF (c1 AND (sa1 OR sa2 OR sa4 OR NOT sa3)) OR (c2 AND (sb1 OR sb2 OR sb4 OR NOT sb3)) THEN
	c3 := TRUE;
	IF (sc1 OR sc2 OR sc4 OR sc3) THEN
		c3:= FALSE;
		e1 := TRUE;
	END_IF
ELSE
	c3:= FALSE;
END_IF

q1 := c1 AND NOT sa1;
q2 := c2 AND NOT sa2;
q3 := c3 AND NOT sa3;


IF phaselock THEN
q1:=FALSE;
q2:=FALSE;
q3:=FALSE;
END_IF
END_FUNCTION_BLOCK

(* POU EQUIP_TYPE_11, ST *)
FUNCTION_BLOCK EQUIP_TYPE_11

VAR_INPUT
	i1 : BOOL;
	i2 : BOOL;

	sa1 : BOOL;
	sa2 : BOOL;

END_VAR
VAR_OUTPUT
	c1 : BOOL;
	q1 : BOOL;
	e1 : BOOL;
END_VAR
VAR
END_VAR
c1 := (i2 OR c1) AND NOT i1;
e1 :=( ( sa1 OR sa2));
q1 := c1;


IF phaselock THEN
q1:=FALSE;
END_IF
END_FUNCTION_BLOCK

(* POU Reactor, ST *)
FUNCTION_BLOCK Reactor
VAR_INPUT
	op: BOOL;
	res_fill: BOOL;
	i1: BOOL;
	alum_time: TIME := T#5s;
	res_aeration: BOOL;
	ph1: REAL;
	res_decanting: BOOL;
	r1: BOOL;
	i2: BOOL;
	i3: BOOL;
	i4: BOOL;
	reset : BOOL;
END_VAR
VAR_OUTPUT
	req_fill: BOOL;
	q1: BOOL;
	q2: BOOL;
	q4: BOOL;
	q3: BOOL;
	q5: BOOL;
	q6: BOOL;
	req_aeration: BOOL;
	e1: BOOL;
	q7: BOOL;
	q8: BOOL;
	m1:BOOL;
	req_settle: BOOL;
	req_decanting: BOOL;
	q9: BOOL;
END_VAR
VAR
	TON1: TON;
	TP1: TP;
	TON2: TON;
	TON3: TON;
	decanting_done: BOOL;
	start_decanter: BOOL;
	TON4: TON;
	decanter: INT;
	TP2: TP;
	TP3: TP;
END_VAR
VAR PERSISTENT
	seq: INT;
END_VAR
IF reset THEN
seq := 0;
END_IF


req_fill := FALSE;
req_aeration := FALSE;
req_settle:= FALSE;
req_decanting := FALSE;
start_decanter := FALSE;
q1 := FALSE;
q2 := FALSE;
q3 := FALSE;
q4 := FALSE;
q5 := FALSE;

q6 := FALSE;
q7 := FALSE;

q8 := FALSE;
q9 := FALSE;
CASE seq OF
0:
	IF op THEN
		seq := 1;
	END_IF
1:
IF op THEN
	req_fill := TRUE;
	q1 := res_fill;
	q2 := res_fill;

	IF i1 THEN
		seq := 2;
	END_IF
ELSE
	seq := 0;
END_IF
2:
IF op THEN
	req_aeration := TRUE;
	IF res_aeration THEN
		TON2(IN:= TRUE,PT:=T#3.5h , Q=> , ET=> );

		TON1(IN:= TRUE, PT:=T#2h , Q=> e1, ET=> );
		TP1(IN:=TON1.Q AND r1 , PT:=alum_time , Q=>q4 , ET=> );
		q5 := TRUE;
		m1 := ((m1 OR (ph1 <= 5)) AND ph1 > 7.5);
		q3 := m1;
		IF ton2.Q THEN
			TON2(IN:= FALSE,PT:=T#3.5h , Q=> , ET=> );

			TON1(IN:= FALSE, PT:=T#2h , Q=> e1, ET=> );
			TP1(IN:=FALSE , PT:=alum_time , Q=>q4 , ET=> );
			seq := 3;
		END_IF
	END_IF

ELSE
	seq := 0;
	TON2(IN:= FALSE,PT:=T#3.5h , Q=> , ET=> );

	TON1(IN:= FALSE, PT:=T#2h , Q=> e1, ET=> );
	TP1(IN:=FALSE , PT:=alum_time , Q=>q4 , ET=> );
END_IF
3:
IF op THEN
	req_settle  := TRUE;
	TON3(IN:=TRUE ,  PT:=T#1.5h);
	IF ton3.Q THEN
		seq:= 4;
		TON3(IN:=FALSE ,  PT:=T#1.5h);
	END_IF
ELSE
	seq:= 0;
	TON3(IN:=FALSE ,  PT:=T#1.5h);
END_IF

4:
IF op THEN
 	req_decanting := TRUE;
	IF res_decanting THEN
		start_decanter := TRUE;
	END_IF
	IF decanting_done THEN
		seq := 0;
		TON4(IN:=FALSE ,  PT:=T#3606s);
	END_IF
	TON4(IN:=TRUE, PT:=T#3606s);
	IF ((TON4.ET < T#15m) OR (TON4.ET > T#45m)) AND NOT i2 THEN
		q6 := TRUE;
		q7 := TRUE;
	END_IF
ELSE
	seq:=0;
END_IF
END_CASE


decanting_done := FALSE;
CASE decanter OF
0:
	q8 := NOT i3;
	q9 := FALSE;

	IF i3 AND start_decanter THEN
		decanter := 1;
	END_IF

1:
	q8 := FALSE;
	IF start_decanter THEN
		TP2(IN:=TRUE , PT:=T#45s , Q=> q9, ET=> );
		IF NOT TP2.Q OR i4 THEN
			decanter := 2;
			TP2(IN:=FALSE , PT:=T#45s , Q=> q9, ET=> );
		END_IF
	END_IF
2:
	IF start_decanter THEN
		TP3(IN:=TRUE , PT:=T#5s , Q=> q9, ET=> );
		IF i4 THEN
			decanter := 4;
			TP3(IN:=FALSE , PT:=T#5s , Q=> q9, ET=> );
		ELSIF (NOT TP3.Q) THEN
			decanter := 1;
			TP3(IN:=FALSE , PT:=T#5s , Q=> q9, ET=> );
		END_IF
	END_IF
4:
	q8 := NOT i3;
	q9 := FALSE;
	IF i3 THEN
		decanting_done := TRUE;
		decanter := 0;
	END_IF

END_CASE
END_FUNCTION_BLOCK

(* POU timeConversion, ST *)
FUNCTION_BLOCK timeConversion
VAR_INPUT
	inputTime : WORD;
END_VAR
VAR_OUTPUT
	outputTime : WORD;
END_VAR
VAR
	inputTimeOTSTRUCT : OTSTRUCT;
	outputTimeOTSTRUCT : OTSTRUCT;
END_VAR
VAR_IN_OUT
	atTime : TIME;
END_VAR
inputTimeOTSTRUCT.wSecond := inputTime;
atTime := OTSTRUCT_TO_TIME(inputTimeOTSTRUCT);

outputTimeOTSTRUCT := TIME_TO_OTSTRUCT(atTime);
outputTime:= outputTimeOTSTRUCT.wSecond + (outputTimeOTSTRUCT.wMinute * 60) + (outputTimeOTSTRUCT.wHour * 60 * 60) + (outputTimeOTSTRUCT.wDay * 60 *60 *24);
END_FUNCTION_BLOCK

(* POU Fill_selector, ST *)
FUNCTION_BLOCK Fill_selector
VAR_INPUT
	i1: BOOL;
	i2: BOOL;
	i3: BOOL;
	i4: BOOL;
END_VAR
VAR_OUTPUT
	q1: BOOL;
	q2: BOOL;
	q3: BOOL;
	q4: BOOL;
	c1 : BOOL;
END_VAR
VAR
	ireactor: INT;
END_VAR
q1 := q2 := q3 := q4 := FALSE;

CASE ireactor OF
0:
	IF NOT i1 THEN
		ireactor := 1;
	END_IF
	q1 := TRUE;
1:
	IF NOT i2 THEN
		ireactor := 2;
	END_IF
	q2 := TRUE;
2:
	IF NOT i3 THEN
		ireactor := 3;
	END_IF
	q3 := TRUE;
3:
	IF NOT i4 THEN
		ireactor := 0;
	END_IF
	q4 := TRUE;
END_CASE

c1 := i1 OR i2 OR i3 OR i4;
END_FUNCTION_BLOCK

(* POU blower_selector, ST *)
FUNCTION_BLOCK blower_selector
VAR_INPUT
	i1 :BOOL;
	i2: BOOL;
	i3 : BOOL;
	i4 : BOOL;
	available : INT;
END_VAR
VAR_OUTPUT
	q1 : BOOL;
	q2 : BOOL;
	q3 : BOOL;
	q4 : BOOL;
	taken : INT;
END_VAR
VAR
	request: ARRAY [1..4] OF BOOL;
	respond: ARRAY [1..4] OF BOOL;
	b: INT;
	a: INT;
END_VAR
request[a];
respond[b];
taken;
available;


request[1] := i1;
request[2] := i2;
request[3] := i3;
request[4] := i4;
FOR a:= 1 TO 4 DO
IF request[a] AND NOT respond[a] THEN
	IF available - taken > 0 THEN
		respond[a] := TRUE;
		taken := taken+ 1;
	END_IF
END_IF
END_FOR

FOR b:=1 TO 4 DO
IF respond[b] THEN
	IF NOT request[b] THEN
		respond[b] := FALSE;
		taken := taken -1;
		IF taken < 0 THEN
			taken := 0;
		END_IF
	END_IF
END_IF
END_FOR
q1 := respond[1];
q2 := respond[2];
q3 := respond[3];
q4 := respond[4];
END_FUNCTION_BLOCK

(* POU Decant_selector, ST *)
FUNCTION_BLOCK Decant_selector
VAR_INPUT
	i1: BOOL;
	i2: BOOL;
	i3: BOOL;
	i4: BOOL;
END_VAR
VAR_OUTPUT
	q1: BOOL;
	q2: BOOL;
	q3: BOOL;
	q4: BOOL;
	c1: BOOL;
END_VAR
VAR
	ireactor: INT;
END_VAR
q1 := q2 := q3 := q4 := FALSE;

CASE ireactor OF
0:
	IF NOT i1 THEN
		ireactor := 1;
	END_IF
	q1 := TRUE;
1:
	IF NOT i2 THEN
		ireactor := 2;
	END_IF
	q2 := TRUE;
2:
	IF NOT i3 THEN
		ireactor := 3;
	END_IF
	q3 := TRUE;
3:
	IF NOT i4 THEN
		ireactor := 0;
	END_IF
	q4 := TRUE;
END_CASE

c1 := i1 OR i2 OR i3 OR i4;
END_FUNCTION_BLOCK

(* POU EQUIP_TYPE_9, ST *)
FUNCTION_BLOCK EQUIP_TYPE_9 (*valve with 2 output*)
VAR_INPUT
	i1:BOOL;
	i2 : BOOL;
	s1:BOOL;
	s2:BOOL;
END_VAR
VAR_OUTPUT
	c1 : BOOL;
	q1: BOOL;
	q2: BOOL;
	e1:BOOL;
END_VAR
VAR
END_VAR
c1 := (i2 OR c1) AND NOT i1;
q1 := NOT c1;
q2 := c1;


IF phaselock THEN
q1:=FALSE;
q2:=FALSE;
END_IF
END_FUNCTION_BLOCK

(* POU EQUIP_TYPE_8, ST *)
FUNCTION_BLOCK EQUIP_TYPE_8 (*3 EQUIPMENT START AT THE SAME TIME*)
VAR_INPUT
	i1 : BOOL;
	i2 : BOOL;


	sa1 : BOOL;
	sa2 : BOOL;
	sa3 : BOOL;
	sa4 : BOOL;
	sa5 : BOOL;

	sb1 : BOOL;
	sb2 : BOOL;
	sb3 : BOOL;
	sb4 : BOOL;
	sb5 : BOOL;

	sc1 : BOOL;
	sc2 : BOOL;
	sc3 : BOOL;
	sc4 : BOOL;
	sc5 : BOOL;
END_VAR
VAR_OUTPUT
	c1 : BOOL;
	q1 : BOOL;
	q2 : BOOL;
	q3 : BOOL;
	e1 : BOOL;
END_VAR
VAR
END_VAR
c1 := (i2 OR c1) AND NOT i1;
e1 :=(( (sa2 OR sa4 OR sa1) AND (sb2 OR sb4 OR sb1)AND (sc2 OR sc4 OR sc1)));
q1 := c1 AND NOT sa3;
q2 := c1 AND NOT sb3;
q3 := c1 AND NOT sc3;


IF phaselock THEN
q1:=FALSE;
q2:=FALSE;
q3:=FALSE;
END_IF
END_FUNCTION_BLOCK

(* POU EQUIP_TYPE_10, ST *)
FUNCTION_BLOCK EQUIP_TYPE_10
VAR_INPUT
	i1:BOOL;
	i2:BOOL;
	r1:BOOL;
	s1:BOOL;
	s2:BOOL;
	s3:BOOL;
	s4:BOOL;
	s5:BOOL;

END_VAR
VAR_OUTPUT
	q1:BOOL;
	q2:BOOL;
	e1:BOOL;
END_VAR
VAR
END_VAR
q1 := i1;
q2 := i2;


IF phaselock THEN
q1:=FALSE;
q2:=FALSE;
END_IF
END_FUNCTION_BLOCK

(* POU EQUIPMENT_SBR_AIRBLOWER, ST *)
FUNCTION_BLOCK EQUIPMENT_SBR_AIRBLOWER
VAR_INPUT
	sa1 : BOOL;
	sa2 : BOOL;
	sa3 : BOOL;
	sa4 : BOOL;
	sa5 : BOOL;

	sb1 : BOOL;
	sb2 : BOOL;
	sb3 : BOOL;
	sb4 : BOOL;
	sb5 : BOOL;

	sc1 : BOOL;
	sc2 : BOOL;
	sc3 : BOOL;
	sc4 : BOOL;
	sc5 : BOOL;
	req : INT;
	r1: BOOL;
	hold : BOOL;


END_VAR
VAR_OUTPUT
	rq1 : BOOL;
	rq2 : BOOL;
	rq3 : BOOL;
	e1: BOOL;
	e2: BOOL;
	e3: BOOL;
	res :  INT;
	e: BOOL;
END_VAR
VAR
	q1 : BOOL;
	q2 : BOOL;
	q3 : BOOL;

	pump1: INT;
	rest1: BOOL;
	TONOFF1: TON;
	decommission: BOOL;
	TONON1: TON;
	Count_bool1: Count_bool;
	pump2: INT;
	TONON2: TON;
	TONOFF2: TON;
	rest2: BOOL;
	pump3: INT;
	TONOFF3: TON;
	rest3: BOOL;
	TONON3: TON;
END_VAR
CASE pump1 OF
0:
	TONOFF1( PT:=t#10m , Q=> , ET=> );
	IF tonoff1.Q THEN
		rest1 := FALSE;
	END_IF
		q1 := FALSE;
 	IF (req > res) AND NOT rest1 AND NOT e1 THEN
		pump1 := 1;
		q1 := TRUE;
		TONOFF1(IN:=FALSE , PT:=t#10m , Q=> , ET=> );
	END_IF
1:
	TONON1(IN:= TRUE, PT:=T#1h10m , Q=> , ET=> );
	IF TONON1.Q OR e1 OR decommission THEN
		decommission := FALSE;
		TONON1(IN:= FALSE, PT:=T#1h10m , Q=> , ET=> );
		TONOFF1(IN:=TRUE , PT:=t#10m , Q=> , ET=> );
		rest1:= TRUE;
		pump1 := 0;
	END_IF
END_CASE


CASE pump2 OF
0:
	TONOFF2( PT:=t#10m , Q=> , ET=> );
	IF tonoff2.Q THEN
		rest2 := FALSE;
	END_IF
		q2 := FALSE;
 	IF (req > res) AND NOT rest2 AND NOT e2 THEN
		pump2 := 1;
		q2:= TRUE;
		TONOFF2(IN:=FALSE , PT:=t#10m , Q=> , ET=> );
	END_IF
1:
	TONON2(IN:= TRUE, PT:=T#1h10m , Q=> , ET=> );
	IF TONON2.Q OR e2 OR decommission THEN
		decommission := FALSE;
		TONON2(IN:= FALSE, PT:=T#1h10m , Q=> , ET=> );
		TONOFF2(IN:=TRUE , PT:=t#10m , Q=> , ET=> );
		rest2:= TRUE;
		pump2 := 0;
	END_IF
END_CASE

CASE pump3 OF
0:
	TONOFF3( PT:=t#10m , Q=> , ET=> );
	IF tonoff3.Q THEN
		rest3 := FALSE;
	END_IF
		q3 := FALSE;
 	IF (req > res) AND NOT rest3 AND NOT e3 THEN
		pump3 := 1;
		q3:= TRUE;
		TONOFF3(IN:=FALSE , PT:=t#10m , Q=> , ET=> );
	END_IF
1:
	TONON3(IN:= TRUE, PT:=T#1h10m , Q=> , ET=> );
	IF TONON3.Q OR e3 OR decommission THEN
		decommission := FALSE;
		TONON3(IN:= FALSE, PT:=T#1h10m , Q=> , ET=> );
		TONOFF3(IN:=TRUE , PT:=t#10m , Q=> , ET=> );
		rest3:= TRUE;
		pump3 := 0;
	END_IF
END_CASE


e1 := sa1 OR sa2 OR sa3 OR sa4;
e2 := sb1 OR sb2 OR sb3 OR sb4;
e3 := sc1 OR sc2 OR sc3 OR sc4;

e:= (((e1 AND NOT sa3) AND (e2 AND NOT sb3) AND (e3 AND NOT sc3)) OR e) AND NOT r1;

IF e THEN
pump1 := 0;
pump2 := 0;
pump3 := 0;
END_IF


Count_bool1(
	i1:=q1 ,
	i2:= q2,
	i3:= q3,
	i4:= FALSE,
	q=> res);

IF req < res THEN
decommission := TRUE;
END_IF

rq1 := q1 AND NOT hold;
rq2 := q2 AND NOT hold;
rq3 := q3 AND NOT hold;


IF phaselock THEN
q1:=FALSE;
q2:=FALSE;
q3:=FALSE;

rq1:=FALSE;
rq2:=FALSE;
rq3:=FALSE;
END_IF
END_FUNCTION_BLOCK

(* POU Count_bool, ST *)
FUNCTION_BLOCK Count_bool
VAR_INPUT
	i1 : BOOL;
	i2 : BOOL;
	i3: BOOL;
	i4 : BOOL;
END_VAR
VAR_OUTPUT
	q:INT;
END_VAR
VAR
END_VAR
q := 0;
IF i1 THEN
	q:= q + 1;
END_IF
IF i2 THEN
	q:= q + 1;
END_IF
IF i3 THEN
	q:= q + 1;
END_IF
IF i4 THEN
	q:= q + 1;
END_IF
END_FUNCTION_BLOCK

(* POU sludge_holding, ST *)
FUNCTION_BLOCK sludge_holding
VAR_INPUT
	i1A : BOOL;
	i1B : BOOL;
	i2A : BOOL;
	i2B : BOOL;
	i3A : BOOL;
	i3B : BOOL;
	i4 : BOOL;
	i5 : BOOL;
	i6 : BOOL;
	i7 : BOOL;
	ic1 : BOOL;
	ic2 : BOOL;
	if1: BOOL;
	if2: BOOL;
	sb1: BOOL;
	sbs1: BOOL;
	s1 : BOOL;
	s2 : BOOL;
	s3 : BOOL;
	s4 : BOOL;
	s5 : BOOL;
	r1 : BOOL;


END_VAR
VAR_OUTPUT
	q1A : BOOL;
	q2A : BOOL;
	q1B : BOOL;
	q2B : BOOL;
	q3 : BOOL;
	q4 : BOOL;
	q5 : BOOL;
	q6 : BOOL;
	q7 : BOOL;
	q8 : BOOL;
	q9_1A:BOOL;
	q9_2A:BOOL;
	q9_1B:BOOL;
	q9_2B:BOOL;
	q10 : BOOL;
	q11 : BOOL;
	q12 : BOOL;
	q13 : BOOL;
	q14 : BOOL;
	pfa1: BOOL;
	pfa2: BOOL;
	c1 : BOOL;
	e1 : BOOL;

END_VAR
VAR
	TON1 : TON;
	TOF1 : TOF;
END_VAR
q9_1A := q1A := NOT i1A;
q9_2A := q2A := i2A;

q9_1B := q1B := NOT i1B;
q9_2B := q2B := i2B;

(*single switch convention*)
q3 := ic1 AND s4;
q4 := ic2 AND s5;

(* t /ops *)
c1 := (i2A OR i2B OR c1) AND NOT ((NOT i1A AND NOT i2A) OR s1 OR s2 OR s3 OR i7);

TON1(IN:=i4 , PT:=T#3s , Q=> , ET=> );
(*single switch*)
q5 := c1;
q6 := c1 AND TON1.Q;
q7 := c1;
q8 := c1;


q10 := i5;
q11 := (NOT i6) AND r1;
e1 := (e1 OR i6) AND NOT r1;
q12 := i6;

TOF1(IN:=i6 , PT:=T#30s , Q=> , ET=> );
q14 := q13 := c1 AND TOF1.Q;


(* filterate sump *)
pfa1 := if1 OR sb1;
pfa2 := if2 AND sbs1 AND (NOT sb1);
END_FUNCTION_BLOCK

(* POU EQUIP_STIRRER, ST *)
FUNCTION_BLOCK EQUIP_STIRRER
(*
	sa1:= F101B2_FineScr_EStopStat,
	sa2:= F101B2_FineScr_LocalRemoteStat,
	sa3:= F101B2_FineScr_OverloadStat,
	sa4:= F101B2_FineScr_RunStat,
*)
VAR_INPUT
	i1 : BOOL;
	i2 : BOOL;

	sa1 : BOOL;
	sa2 : BOOL;
	sa3 : BOOL;
	sa4 : BOOL;

END_VAR
VAR_OUTPUT
	c1 : BOOL;
	q1 : BOOL;
	q2 : BOOL;
	e1 : BOOL;
END_VAR
VAR
	stir: INT;
	backward: BOOL;
	TON1: TON;
	forward: BOOL;
END_VAR
c1 := (i2 OR c1) AND NOT i1;
e1 :=( ( sa3 OR sa1));
q1 := c1 AND forward;
q2 := c1 AND backward;

IF NOT c1 THEN
	stir := 0;
	TON1(IN:=FALSE , PT:=T#30s , Q=> , ET=> );
END_IF


CASE stir OF
0 :
	forward:=FALSE;
	backward := TRUE;
	TON1(IN:=TRUE , PT:=T#5m , Q=> , ET=> );
	IF ton1.Q THEN
	TON1(IN:=FALSE , PT:=T#5m , Q=> , ET=> );
	stir := 1;
	END_IF
1:
	backward := FALSE;
	forward := FALSE;
	TON1(IN:=TRUE , PT:=T#30s , Q=> , ET=> );
	IF ton1.Q THEN
	TON1(IN:=FALSE , PT:=T#30s , Q=> , ET=> );
	stir := 2;
	END_IF
2:
	forward:=TRUE;
	backward := FALSE;
	TON1(IN:=TRUE , PT:=T#5m , Q=> , ET=> );
	IF ton1.Q THEN
	TON1(IN:=FALSE , PT:=T#5m , Q=> , ET=> );
	stir := 0;
	END_IF
END_CASE

IF sa2 THEN
forward := FALSE;
backward := FALSE;
END_IF;

IF phaselock THEN
q1:=FALSE;
q2:=FALSE;
END_IF
END_FUNCTION_BLOCK

(* POU tertiary_treatment_plant, ST *)
FUNCTION_BLOCK tertiary_treatment_plant
VAR_INPUT
	i1 : BOOL;
	i2 : BOOL;
	i3 : BOOL;
	i4 : BOOL;
	i5 : BOOL;
	i6 : BOOL;
	i7 : BOOL;
	s1 : BOOL;
	s2 : BOOL;
	s3 : BOOL;
	s4 : BOOL;
END_VAR
VAR_OUTPUT
	q1: BOOL;
	q2 : BOOL;
	q3 : BOOL;
	q4 : BOOL;
	q5 : BOOL;
	q6 : BOOL;
	q7 : BOOL;
	q8 : BOOL;
	q9 : BOOL;
	q10 : BOOL;
	q11 : BOOL;
	q12 : BOOL;
END_VAR
VAR
END_VAR
q1 := i3 OR i4;
q2 := i1 OR NOT i4;
q3:= NOT(s3 OR s4);
q4 := (s3 OR s4);
q5 := NOT(s3 OR s4);
q6 := (s3 OR s4);
q7 := NOT ( s1 OR s2);
q8 := (s1 OR s2);
q9:= NOT i5;
q10 := i5;
q11 := i7 OR NOT(s1 OR s2);
q12 := NOT i6 AND (s1 OR s2);
END_FUNCTION_BLOCK

(* POU EQUIP_TYPE_12, ST *)
FUNCTION_BLOCK EQUIP_TYPE_12 (*5 min per hour*)
VAR_INPUT
	i1 : BOOL;
	i2 : BOOL;

	sa1 : BOOL;
	sa2 : BOOL;

END_VAR
VAR_OUTPUT
	c1 : BOOL;
	q1 : BOOL;
	e1 : BOOL;
END_VAR
VAR
	timer1: TON;
	timer2: TON;
END_VAR
c1 := (i2 OR c1) AND NOT i1;
q1 := c1 AND NOT timer1.Q;
timer1(IN:=c1 AND NOT timer2.Q , PT:=t#5m , Q=> , ET=> );
timer2(IN:=timer1.Q , PT:=t#1h , Q=> , ET=> );


IF phaselock THEN
q1:=FALSE;
END_IF
END_FUNCTION_BLOCK

(* POU REUSE_WATER, ST *)
FUNCTION_BLOCK REUSE_WATER
VAR_INPUT
	i3: BOOL;
	i1: BOOL;
	i4: BOOL;
	i2: BOOL;
	i5: BOOL;
	i6: BOOL;
	p1: REAL;


END_VAR
VAR_OUTPUT
	q1: BOOL;
	q2: BOOL;
	q3: BOOL;
	q4: BOOL;
	q5: BOOL;
	q6: BOOL;
	q7: BOOL;
	q8: BOOL;
	q9: BOOL;
END_VAR
VAR
	m1: BOOL;
	e1: BOOL;
	TON1: TON;
	m2: BOOL;
	TON2: TON;
END_VAR
q1 := (p1 > 8) OR (NOT m1) OR e1 OR i3;
q2 := (p1 <= 6) AND m1;

q3:=(p1 > 6.4) OR (NOT m1) OR e1 OR i3;
q4 := (p1 <= 5.2) AND m1;

q5:=(p1 > 5.9) OR (NOT m1) OR e1 OR i3;
q6 := (p1 <= 4.7) AND m1;

TON1(IN:=((p1 < 3.5) AND m1) , PT:=T#5s , Q=>e1 , ET=> );
TON2(IN:=i1 , PT:=T#5s , Q=> , ET=> );
m2 := TON2.Q    (*(i2 OR m2) AND i1*);
m1 := i4 AND m2;

q7 := i6;
q8 := i5;

q9 := TRUE;
END_FUNCTION_BLOCK
